LIN {X 0,Y 171.438,Z 260.68,A -85,B 0,C 180,E1 -22896.744,E2 -22896.744} C_VEL
LIN {X 0,Y 171.589,Z 261.495,A -85,B 0,C 180,E1 -22897.442,E2 -22897.442} C_VEL
LIN {X 0,Y 173.16,Z 264.453,A -85,B 0,C 180,E1 -22898.399,E2 -22898.399} C_VEL
LIN {X 0,Y 175.194,Z 266.321,A -85,B 0,C 180,E1 -22899.355,E2 -22899.355} C_VEL
LIN {X 0,Y 177.399,Z 269.743,A -85,B 0,C 180,E1 -22900.432,E2 -22900.432} C_VEL
LIN {X 0,Y 178.724,Z 271.306,A -85,B 0,C 180,E1 -22901.026,E2 -22901.026} C_VEL
LIN {X 0,Y 182.403,Z 276.687,A -85,B 0,C 180,E1 -22902.654,E2 -22902.654} C_VEL
LIN {X 0,Y 187.646,Z 284.442,A -85,B 0,C 180,E1 -22904.791,E2 -22904.791} C_VEL
LIN {X 0,Y 194.854,Z 296.389,A -85,B 0,C 180,E1 -22907.491,E2 -22907.491} C_VEL
LIN {X 0,Y 202.104,Z 310.594,A -85,B 0,C 180,E1 -22910.01,E2 -22910.01} C_VEL
LIN {X 0,Y 211.221,Z 330.235,A -85,B 0,C 180,E1 -22912.895,E2 -22912.895} C_VEL
LIN {X 0,Y 219.903,Z 344.859,A -85,B 0,C 180,E1 -22915.172,E2 -22915.172} C_VEL
LIN {X 0,Y 228.476,Z 356.909,A -85,B 0,C 180,E1 -22917.153,E2 -22917.153} C_VEL
LIN {X 0,Y 236.72,Z 367.005,A -85,B 0,C 180,E1 -22919.009,E2 -22919.009} C_VEL
LIN {X 0,Y 244.162,Z 375.394,A -85,B 0,C 180,E1 -22920.704,E2 -22920.704} C_VEL
LIN {X 0,Y 253.065,Z 384.472,A -85,B 0,C 180,E1 -22922.707,E2 -22922.707} C_VEL
LIN {X 0,Y 263.679,Z 393.909,A -85,B 0,C 180,E1 -22924.986,E2 -22924.986} C_VEL
LIN {X 0,Y 276.755,Z 403.951,A -85,B 0,C 180,E1 -22927.61,E2 -22927.61} C_VEL
LIN {X 0,Y 290.97,Z 414.153,A -85,B 0,C 180,E1 -22930.386,E2 -22930.386} C_VEL
LIN {X 0,Y 299.98,Z 420.738,A -85,B 0,C 180,E1 -22932.268,E2 -22932.268} C_VEL
LIN {X 0,Y 305.133,Z 424.274,A -85,B 0,C 180,E1 -22933.436,E2 -22933.436} C_VEL
LIN {X 0,Y 312.329,Z 429.408,A -85,B 0,C 180,E1 -22935.367,E2 -22935.367} C_VEL
LIN {X 0,Y 318.737,Z 433.404,A -85,B 0,C 180,E1 -22937.262,E2 -22937.262} C_VEL
LIN {X 0,Y 322.774,Z 436.101,A -85,B 0,C 180,E1 -22938.699,E2 -22938.699} C_VEL
LIN {X 0,Y 327.517,Z 439.409,A -85,B 0,C 180,E1 -22940.778,E2 -22940.778} C_VEL
LIN {X 0,Y 331.24,Z 441.589,A -85,B 0,C 180,E1 -22942.686,E2 -22942.686} C_VEL
LIN {X 0,Y 333.408,Z 442.651,A -85,B 0,C 180,E1 -22943.95,E2 -22943.95} C_VEL
LIN {X 0,Y 335.133,Z 443.443,A -85,B 0,C 180,E1 -22945.188,E2 -22945.188} C_VEL
LIN {X 0,Y 336.579,Z 443.963,A -85,B 0,C 180,E1 -22946.409,E2 -22946.409} C_VEL
LIN {X 0,Y 337.607,Z 444.405,A -85,B 0,C 180,E1 -22947.718,E2 -22947.718} C_VEL
LIN {X 0,Y 338.329,Z 444.651,A -85,B 0,C 180,E1 -22950,E2 -22950} C_VEL
LIN {X 0,Y 338.048,Z 444.627,A -85,B 0,C 180,E1 -22951.191,E2 -22951.191} C_VEL
LIN {X 0,Y 337.557,Z 444.334,A -85,B 0,C 180,E1 -22952.386,E2 -22952.386} C_VEL
LIN {X 0,Y 336.548,Z 443.959,A -85,B 0,C 180,E1 -22953.592,E2 -22953.592} C_VEL
LIN {X 0,Y 335.114,Z 443.428,A -85,B 0,C 180,E1 -22954.812,E2 -22954.812} C_VEL
LIN {X 0,Y 332.51,Z 442.258,A -85,B 0,C 180,E1 -22956.593,E2 -22956.593} C_VEL
LIN {X 0,Y 327.517,Z 439.388,A -85,B 0,C 180,E1 -22959.222,E2 -22959.222} C_VEL
LIN {X 0,Y 322.58,Z 435.992,A -85,B 0,C 180,E1 -22961.364,E2 -22961.364} C_VEL
LIN {X 0,Y 318.737,Z 433.444,A -85,B 0,C 180,E1 -22962.738,E2 -22962.738} C_VEL
LIN {X 0,Y 312.33,Z 429.414,A -85,B 0,C 180,E1 -22964.633,E2 -22964.633} C_VEL
LIN {X 0,Y 307.142,Z 425.748,A -85,B 0,C 180,E1 -22966.049,E2 -22966.049} C_VEL
LIN {X 0,Y 301.836,Z 422,A -85,B 0,C 180,E1 -22967.324,E2 -22967.324} C_VEL
LIN {X 0,Y 293.695,Z 416.255,A -85,B 0,C 180,E1 -22969.055,E2 -22969.055} C_VEL
LIN {X 0,Y 282.709,Z 408.344,A -85,B 0,C 180,E1 -22971.217,E2 -22971.217} C_VEL
LIN {X 0,Y 267.705,Z 397.193,A -85,B 0,C 180,E1 -22974.18,E2 -22974.18} C_VEL
LIN {X 0,Y 255.704,Z 386.898,A -85,B 0,C 180,E1 -22976.717,E2 -22976.717} C_VEL
LIN {X 0,Y 247.803,Z 379.333,A -85,B 0,C 180,E1 -22978.456,E2 -22978.456} C_VEL
LIN {X 0,Y 238.025,Z 368.544,A -85,B 0,C 180,E1 -22980.691,E2 -22980.691} C_VEL
LIN {X 0,Y 229.51,Z 358.161,A -85,B 0,C 180,E1 -22982.64,E2 -22982.64} C_VEL
LIN {X 0,Y 221.548,Z 347.302,A -85,B 0,C 180,E1 -22984.436,E2 -22984.436} C_VEL
LIN {X 0,Y 212.624,Z 332.89,A -85,B 0,C 180,E1 -22986.708,E2 -22986.708} C_VEL
LIN {X 0,Y 204.842,Z 316.83,A -85,B 0,C 180,E1 -22989.069,E2 -22989.069} C_VEL
LIN {X 0,Y 200.046,Z 306.438,A -85,B 0,C 180,E1 -22990.683,E2 -22990.683} C_VEL
LIN {X 0,Y 193.65,Z 294.248,A -85,B 0,C 180,E1 -22992.945,E2 -22992.945} C_VEL
LIN {X 0,Y 186.501,Z 282.617,A -85,B 0,C 180,E1 -22995.666,E2 -22995.666} C_VEL
LIN {X 0,Y 180.746,Z 274.26,A -85,B 0,C 180,E1 -22998.065,E2 -22998.065} C_VEL
LIN {X 0,Y 178.122,Z 270.453,A -85,B 0,C 180,E1 -22999.25,E2 -22999.25} C_VEL
LIN {X 0,Y 175.731,Z 267.409,A -85,B 0,C 180,E1 -23000.361,E2 -23000.361} C_VEL
LIN {X 0,Y 174.815,Z 265.84,A -85,B 0,C 180,E1 -23000.828,E2 -23000.828} C_VEL
LIN {X 0,Y 172.55,Z 263.632,A -85,B 0,C 180,E1 -23001.914,E2 -23001.914} C_VEL
LIN {X 0,Y 171.504,Z 261.178,A -85,B 0,C 180,E1 -23002.721,E2 -23002.721} C_VEL
LIN {X 0,Y 171.432,Z 260.639,A -85,B 0,C 180,E1 -23003.529,E2 -23003.529} C_VEL
LIN {X 0,Y 171.454,Z 260.623,A -85,B 0,C 180,E1 -23009.406,E2 -23009.406} C_VEL
LIN {X 0,Y 171.456,Z 260.598,A -85,B 0,C 180,E1 -23014.393,E2 -23014.393} C_VEL
LIN {X 0,Y 171.576,Z 260.565,A -85,B 0,C 180,E1 -23020.873,E2 -23020.873} C_VEL
LIN {X 0,Y 171.591,Z 260.61,A -85,B 0,C 180,E1 -23025.775,E2 -23025.775} C_VEL
LIN {X 0,Y 171.85,Z 260.526,A -85,B 0,C 180,E1 -23030.586,E2 -23030.586} C_VEL
LIN {X 0,Y 171.819,Z 260.581,A -85,B 0,C 180,E1 -23035.309,E2 -23035.309} C_VEL
LIN {X 0,Y 172.331,Z 260.463,A -85,B 0,C 180,E1 -23040.001,E2 -23040.001} C_VEL
LIN {X 0,Y 171.81,Z 260.584,A -85,B 0,C 180,E1 -23044.694,E2 -23044.694} C_VEL
LIN {X 0,Y 171.844,Z 260.524,A -85,B 0,C 180,E1 -23049.417,E2 -23049.417} C_VEL
LIN {X 0,Y 171.569,Z 260.611,A -85,B 0,C 180,E1 -23054.229,E2 -23054.229} C_VEL
LIN {X 0,Y 171.543,Z 260.569,A -85,B 0,C 180,E1 -23059.56,E2 -23059.56} C_VEL
LIN {X 0,Y 171.463,Z 260.59,A -85,B 0,C 180,E1 -23065.612,E2 -23065.612} C_VEL
LIN {X 0,Y 171.458,Z 260.628,A -85,B 0,C 180,E1 -23070.596,E2 -23070.596} C_VEL
LIN {X 0,Y 171.405,Z 260.744,A -85,B 0,C 180,E1 -23076.39,E2 -23076.39} C_VEL
LIN {X 0,Y 171.537,Z 261.477,A -85,B 0,C 180,E1 -23076.997,E2 -23076.997} C_VEL
LIN {X 0,Y 173.009,Z 264.327,A -85,B 0,C 180,E1 -23077.946,E2 -23077.946} C_VEL
LIN {X 0,Y 175.541,Z 267.445,A -85,B 0,C 180,E1 -23079.183,E2 -23079.183} C_VEL
LIN {X 0,Y 178.493,Z 271.992,A -85,B 0,C 180,E1 -23080.599,E2 -23080.599} C_VEL
LIN {X 0,Y 182.943,Z 279.543,A -85,B 0,C 180,E1 -23082.618,E2 -23082.618} C_VEL
LIN {X 0,Y 189.539,Z 291.631,A -85,B 0,C 180,E1 -23085.361,E2 -23085.361} C_VEL
LIN {X 0,Y 194.252,Z 301.668,A -85,B 0,C 180,E1 -23087.205,E2 -23087.205} C_VEL
LIN {X 0,Y 199.621,Z 314.742,A -85,B 0,C 180,E1 -23089.216,E2 -23089.216} C_VEL
LIN {X 0,Y 201.158,Z 324.413,A -85,B 0,C 180,E1 -23090.032,E2 -23090.032} C_VEL
LIN {X 0,Y 201.394,Z 328.625,A -85,B 0,C 180,E1 -23090.279,E2 -23090.279} C_VEL
LIN {X 0,Y 199.139,Z 368.462,A -85,B 0,C 180,E1 -23091.638,E2 -23091.638} C_VEL
LIN {X 0,Y 197.78,Z 380.363,A -85,B 0,C 180,E1 -23092.301,E2 -23092.301} C_VEL
LIN {X 0,Y 195.345,Z 393.909,A -85,B 0,C 180,E1 -23093.425,E2 -23093.425} C_VEL
LIN {X 0,Y 192.883,Z 404.427,A -85,B 0,C 180,E1 -23094.66,E2 -23094.66} C_VEL
LIN {X 0,Y 190.357,Z 413.699,A -85,B 0,C 180,E1 -23096.054,E2 -23096.054} C_VEL
LIN {X 0,Y 187.599,Z 422.641,A -85,B 0,C 180,E1 -23097.734,E2 -23097.734} C_VEL
LIN {X 0,Y 184.625,Z 431.165,A -85,B 0,C 180,E1 -23099.71,E2 -23099.71} C_VEL
LIN {X 0,Y 181.879,Z 438.38,A -85,B 0,C 180,E1 -23101.748,E2 -23101.748} C_VEL
LIN {X 0,Y 179.461,Z 444.58,A -85,B 0,C 180,E1 -23103.86,E2 -23103.86} C_VEL
LIN {X 0,Y 176.889,Z 451.12,A -85,B 0,C 180,E1 -23106.59,E2 -23106.59} C_VEL
LIN {X 0,Y 174.917,Z 455.619,A -85,B 0,C 180,E1 -23108.801,E2 -23108.801} C_VEL
LIN {X 0,Y 172.575,Z 461.112,A -85,B 0,C 180,E1 -23112.216,E2 -23112.216} C_VEL
LIN {X 0,Y 170.821,Z 465.44,A -85,B 0,C 180,E1 -23115.709,E2 -23115.709} C_VEL
LIN {X 0,Y 170.017,Z 467.812,A -85,B 0,C 180,E1 -23118.072,E2 -23118.072} C_VEL
LIN {X 0,Y 169.418,Z 469.615,A -85,B 0,C 180,E1 -23120.449,E2 -23120.449} C_VEL
LIN {X 0,Y 168.933,Z 472.074,A -85,B 0,C 180,E1 -23125.227,E2 -23125.227} C_VEL
LIN {X 0,Y 168.87,Z 472.72,A -85,B 0,C 180,E1 -23128.402,E2 -23128.402} C_VEL
LIN {X 0,Y 168.968,Z 472.826,A -85,B 0,C 180,E1 -23130,E2 -23130} C_VEL
LIN {X 0,Y 168.853,Z 472.607,A -85,B 0,C 180,E1 -23132.627,E2 -23132.627} C_VEL
LIN {X 0,Y 168.863,Z 472.072,A -85,B 0,C 180,E1 -23134.775,E2 -23134.775} C_VEL
LIN {X 0,Y 169.207,Z 470.166,A -85,B 0,C 180,E1 -23138.609,E2 -23138.609} C_VEL
LIN {X 0,Y 168.941,Z 468.894,A -85,B 0,C 180,E1 -23140.562,E2 -23140.562} C_VEL
LIN {X 0,Y 167.041,Z 466.261,A -85,B 0,C 180,E1 -23143.759,E2 -23143.759} C_VEL
LIN {X 0,Y 165.575,Z 462.945,A -85,B 0,C 180,E1 -23146.944,E2 -23146.944} C_VEL
LIN {X 0,Y 165.989,Z 460.535,A -85,B 0,C 180,E1 -23148.811,E2 -23148.811} C_VEL
LIN {X 0,Y 168.79,Z 454.39,A -85,B 0,C 180,E1 -23152.653,E2 -23152.653} C_VEL
LIN {X 0,Y 171.612,Z 447.998,A -85,B 0,C 180,E1 -23155.712,E2 -23155.712} C_VEL
LIN {X 0,Y 174.325,Z 441.439,A -85,B 0,C 180,E1 -23158.275,E2 -23158.275} C_VEL
LIN {X 0,Y 177.779,Z 432.89,A -85,B 0,C 180,E1 -23160.925,E2 -23160.925} C_VEL
LIN {X 0,Y 180.808,Z 424.715,A -85,B 0,C 180,E1 -23162.968,E2 -23162.968} C_VEL
LIN {X 0,Y 183.683,Z 416.208,A -85,B 0,C 180,E1 -23164.69,E2 -23164.69} C_VEL
LIN {X 0,Y 186.22,Z 407.495,A -85,B 0,C 180,E1 -23166.135,E2 -23166.135} C_VEL
LIN {X 0,Y 188.779,Z 397.743,A -85,B 0,C 180,E1 -23167.394,E2 -23167.394} C_VEL
LIN {X 0,Y 190.909,Z 387.666,A -85,B 0,C 180,E1 -23168.405,E2 -23168.405} C_VEL
LIN {X 0,Y 192.614,Z 377.207,A -85,B 0,C 180,E1 -23169.182,E2 -23169.182} C_VEL
LIN {X 0,Y 193.75,Z 367.131,A -85,B 0,C 180,E1 -23169.702,E2 -23169.702} C_VEL
LIN {X 0,Y 195.936,Z 327.052,A -85,B 0,C 180,E1 -23171.126,E2 -23171.126} C_VEL
LIN {X 0,Y 194.539,Z 317.878,A -85,B 0,C 180,E1 -23171.927,E2 -23171.927} C_VEL
LIN {X 0,Y 189.037,Z 304.24,A -85,B 0,C 180,E1 -23174.133,E2 -23174.133} C_VEL
LIN {X 0,Y 184.476,Z 294.52,A -85,B 0,C 180,E1 -23176.044,E2 -23176.044} C_VEL
LIN {X 0,Y 177.798,Z 282.073,A -85,B 0,C 180,E1 -23179.051,E2 -23179.051} C_VEL
LIN {X 0,Y 173.97,Z 275.954,A -85,B 0,C 180,E1 -23180.905,E2 -23180.905} C_VEL
LIN {X 0,Y 171.06,Z 271.361,A -85,B 0,C 180,E1 -23182.419,E2 -23182.419} C_VEL
LIN {X 0,Y 168.608,Z 267.983,A -85,B 0,C 180,E1 -23183.744,E2 -23183.744} C_VEL
LIN {X 0,Y 167.771,Z 266.738,A -85,B 0,C 180,E1 -23184.222,E2 -23184.222} C_VEL
LIN {X 0,Y 165.529,Z 264.614,A -85,B 0,C 180,E1 -23185.464,E2 -23185.464} C_VEL
LIN {X 0,Y 164.434,Z 262.097,A -85,B 0,C 180,E1 -23186.419,E2 -23186.419} C_VEL
LIN {X 0,Y 164.371,Z 261.527,A -85,B 0,C 180,E1 -23187.272,E2 -23187.272} C_VEL
LIN {X 0,Y 164.341,Z 261.476,A -85,B 0,C 180,E1 -23191.937,E2 -23191.937} C_VEL
LIN {X 0,Y 164.412,Z 261.47,A -85,B 0,C 180,E1 -23194.692,E2 -23194.692} C_VEL
LIN {X 0,Y 164.486,Z 261.449,A -85,B 0,C 180,E1 -23200.05,E2 -23200.05} C_VEL
LIN {X 0,Y 164.499,Z 261.486,A -85,B 0,C 180,E1 -23205.146,E2 -23205.146} C_VEL
LIN {X 0,Y 164.765,Z 261.405,A -85,B 0,C 180,E1 -23210.175,E2 -23210.175} C_VEL
LIN {X 0,Y 164.825,Z 261.412,A -85,B 0,C 180,E1 -23212.649,E2 -23212.649} C_VEL
LIN {X 0,Y 165.045,Z 261.392,A -85,B 0,C 180,E1 -23217.558,E2 -23217.558} C_VEL
LIN {X 0,Y 165.293,Z 261.339,A -85,B 0,C 180,E1 -23219.999,E2 -23219.999} C_VEL
LIN {X 0,Y 164.768,Z 261.461,A -85,B 0,C 180,E1 -23224.892,E2 -23224.892} C_VEL
LIN {X 0,Y 164.834,Z 261.419,A -85,B 0,C 180,E1 -23227.347,E2 -23227.347} C_VEL
LIN {X 0,Y 164.703,Z 261.418,A -85,B 0,C 180,E1 -23231.061,E2 -23231.061} C_VEL
LIN {X 0,Y 164.54,Z 261.49,A -85,B 0,C 180,E1 -23234.848,E2 -23234.848} C_VEL
LIN {X 0,Y 164.471,Z 261.452,A -85,B 0,C 180,E1 -23239.988,E2 -23239.988} C_VEL
LIN {X 0,Y 164.383,Z 261.473,A -85,B 0,C 180,E1 -23246.127,E2 -23246.127} C_VEL
LIN {X 0,Y 164.385,Z 261.491,A -85,B 0,C 180,E1 -23252.376,E2 -23252.376} C_VEL
LIN {X 0,Y 164.377,Z 261.818,A -85,B 0,C 180,E1 -23253.765,E2 -23253.765} C_VEL
LIN {X 0,Y 164.717,Z 263.033,A -85,B 0,C 180,E1 -23254.365,E2 -23254.365} C_VEL
LIN {X 0,Y 166.416,Z 265.672,A -85,B 0,C 180,E1 -23255.434,E2 -23255.434} C_VEL
LIN {X 0,Y 168.281,Z 267.143,A -85,B 0,C 180,E1 -23256.427,E2 -23256.427} C_VEL
LIN {X 0,Y 170.322,Z 270.482,A -85,B 0,C 180,E1 -23257.582,E2 -23257.582} C_VEL
LIN {X 0,Y 172.089,Z 272.336,A -85,B 0,C 180,E1 -23258.467,E2 -23258.467} C_VEL
LIN {X 0,Y 174.73,Z 276.02,A -85,B 0,C 180,E1 -23259.785,E2 -23259.785} C_VEL
LIN {X 0,Y 181.065,Z 285.342,A -85,B 0,C 180,E1 -23262.689,E2 -23262.689} C_VEL
LIN {X 0,Y 187.19,Z 295.122,A -85,B 0,C 180,E1 -23265.219,E2 -23265.219} C_VEL
LIN {X 0,Y 192.958,Z 305.583,A -85,B 0,C 180,E1 -23267.427,E2 -23267.427} C_VEL
LIN {X 0,Y 199.509,Z 319.465,A -85,B 0,C 180,E1 -23269.79,E2 -23269.79} C_VEL
LIN {X 0,Y 206.442,Z 334.522,A -85,B 0,C 180,E1 -23272.063,E2 -23272.063} C_VEL
LIN {X 0,Y 215.092,Z 349.3,A -85,B 0,C 180,E1 -23274.448,E2 -23274.448} C_VEL
LIN {X 0,Y 223.821,Z 361.843,A -85,B 0,C 180,E1 -23276.619,E2 -23276.619} C_VEL
LIN {X 0,Y 233.68,Z 374.129,A -85,B 0,C 180,E1 -23279.106,E2 -23279.106} C_VEL
LIN {X 0,Y 244.415,Z 385.978,A -85,B 0,C 180,E1 -23281.798,E2 -23281.798} C_VEL
LIN {X 0,Y 255.3,Z 396.076,A -85,B 0,C 180,E1 -23284.361,E2 -23284.361} C_VEL
LIN {X 0,Y 267.258,Z 405.597,A -85,B 0,C 180,E1 -23286.98,E2 -23286.98} C_VEL
LIN {X 0,Y 280.847,Z 415.193,A -85,B 0,C 180,E1 -23289.782,E2 -23289.782} C_VEL
LIN {X 0,Y 289.662,Z 421.381,A -85,B 0,C 180,E1 -23291.614,E2 -23291.614} C_VEL
LIN {X 0,Y 298.799,Z 427.73,A -85,B 0,C 180,E1 -23293.606,E2 -23293.606} C_VEL
LIN {X 0,Y 305.423,Z 432.473,A -85,B 0,C 180,E1 -23295.338,E2 -23295.338} C_VEL
LIN {X 0,Y 311.032,Z 436.104,A -85,B 0,C 180,E1 -23296.941,E2 -23296.941} C_VEL
LIN {X 0,Y 315.717,Z 438.976,A -85,B 0,C 180,E1 -23298.443,E2 -23298.443} C_VEL
LIN {X 0,Y 320.624,Z 442.508,A -85,B 0,C 180,E1 -23300.531,E2 -23300.531} C_VEL
LIN {X 0,Y 324.682,Z 444.989,A -85,B 0,C 180,E1 -23302.538,E2 -23302.538} C_VEL
LIN {X 0,Y 326.954,Z 446.165,A -85,B 0,C 180,E1 -23303.83,E2 -23303.83} C_VEL
LIN {X 0,Y 328.836,Z 447.066,A -85,B 0,C 180,E1 -23305.096,E2 -23305.096} C_VEL
LIN {X 0,Y 330.825,Z 447.822,A -85,B 0,C 180,E1 -23306.805,E2 -23306.805} C_VEL
LIN {X 0,Y 331.953,Z 448.338,A -85,B 0,C 180,E1 -23308.787,E2 -23308.787} C_VEL
LIN {X 0,Y 332.279,Z 448.347,A -85,B 0,C 180,E1 -23310,E2 -23310} C_VEL
LIN {X 0,Y 331.971,Z 448.319,A -85,B 0,C 180,E1 -23311.213,E2 -23311.213} C_VEL
LIN {X 0,Y 331.432,Z 448.026,A -85,B 0,C 180,E1 -23312.431,E2 -23312.431} C_VEL
LIN {X 0,Y 330.339,Z 447.637,A -85,B 0,C 180,E1 -23313.659,E2 -23313.659} C_VEL
LIN {X 0,Y 328.819,Z 447.054,A -85,B 0,C 180,E1 -23314.904,E2 -23314.904} C_VEL
LIN {X 0,Y 325.667,Z 445.509,A -85,B 0,C 180,E1 -23316.937,E2 -23316.937} C_VEL
LIN {X 0,Y 322.096,Z 443.445,A -85,B 0,C 180,E1 -23318.786,E2 -23318.786} C_VEL
LIN {X 0,Y 319.098,Z 441.471,A -85,B 0,C 180,E1 -23320.148,E2 -23320.148} C_VEL
LIN {X 0,Y 315.637,Z 438.998,A -85,B 0,C 180,E1 -23321.566,E2 -23321.566} C_VEL
LIN {X 0,Y 310.43,Z 435.777,A -85,B 0,C 180,E1 -23323.224,E2 -23323.224} C_VEL
LIN {X 0,Y 305.196,Z 432.342,A -85,B 0,C 180,E1 -23324.726,E2 -23324.726} C_VEL
LIN {X 0,Y 298.774,Z 427.714,A -85,B 0,C 180,E1 -23326.396,E2 -23326.396} C_VEL
LIN {X 0,Y 289.619,Z 421.383,A -85,B 0,C 180,E1 -23328.389,E2 -23328.389} C_VEL
LIN {X 0,Y 278.513,Z 413.636,A -85,B 0,C 180,E1 -23330.688,E2 -23330.688} C_VEL
LIN {X 0,Y 265.442,Z 404.273,A -85,B 0,C 180,E1 -23333.4,E2 -23333.4} C_VEL
LIN {X 0,Y 252.686,Z 393.803,A -85,B 0,C 180,E1 -23336.239,E2 -23336.239} C_VEL
LIN {X 0,Y 242.681,Z 384.19,A -85,B 0,C 180,E1 -23338.632,E2 -23338.632} C_VEL
LIN {X 0,Y 231.94,Z 372.072,A -85,B 0,C 180,E1 -23341.336,E2 -23341.336} C_VEL
LIN {X 0,Y 222.059,Z 359.477,A -85,B 0,C 180,E1 -23343.822,E2 -23343.822} C_VEL
LIN {X 0,Y 212.255,Z 344.794,A -85,B 0,C 180,E1 -23346.29,E2 -23346.29} C_VEL
LIN {X 0,Y 204.9,Z 331.451,A -85,B 0,C 180,E1 -23348.411,E2 -23348.411} C_VEL
LIN {X 0,Y 195.717,Z 311.251,A -85,B 0,C 180,E1 -23351.556,E2 -23351.556} C_VEL
LIN {X 0,Y 189.608,Z 299.314,A -85,B 0,C 180,E1 -23353.839,E2 -23353.839} C_VEL
LIN {X 0,Y 182.777,Z 287.906,A -85,B 0,C 180,E1 -23356.584,E2 -23356.584} C_VEL
LIN {X 0,Y 176.826,Z 279.161,A -85,B 0,C 180,E1 -23359.209,E2 -23359.209} C_VEL
LIN {X 0,Y 174.486,Z 275.766,A -85,B 0,C 180,E1 -23360.328,E2 -23360.328} C_VEL
LIN {X 0,Y 171.432,Z 271.566,A -85,B 0,C 180,E1 -23361.863,E2 -23361.863} C_VEL
LIN {X 0,Y 169.042,Z 268.695,A -85,B 0,C 180,E1 -23363.114,E2 -23363.114} C_VEL
LIN {X 0,Y 167.925,Z 266.813,A -85,B 0,C 180,E1 -23363.762,E2 -23363.762} C_VEL
LIN {X 0,Y 165.577,Z 264.662,A -85,B 0,C 180,E1 -23365.054,E2 -23365.054} C_VEL
LIN {X 0,Y 164.44,Z 262.027,A -85,B 0,C 180,E1 -23366.04,E2 -23366.04} C_VEL
LIN {X 0,Y 164.345,Z 261.512,A -85,B 0,C 180,E1 -23366.924,E2 -23366.924} C_VEL
LIN {X 0,Y 164.401,Z 261.505,A -85,B 0,C 180,E1 -23369.139,E2 -23369.139} C_VEL
LIN {X 0,Y 164.404,Z 261.479,A -85,B 0,C 180,E1 -23374.694,E2 -23374.694} C_VEL
LIN {X 0,Y 164.483,Z 261.45,A -85,B 0,C 180,E1 -23380.053,E2 -23380.053} C_VEL
LIN {X 0,Y 164.54,Z 261.49,A -85,B 0,C 180,E1 -23385.152,E2 -23385.152} C_VEL
LIN {X 0,Y 164.769,Z 261.406,A -85,B 0,C 180,E1 -23390.178,E2 -23390.178} C_VEL
LIN {X 0,Y 164.834,Z 261.419,A -85,B 0,C 180,E1 -23392.653,E2 -23392.653} C_VEL
LIN {X 0,Y 165.049,Z 261.384,A -85,B 0,C 180,E1 -23397.561,E2 -23397.561} C_VEL
LIN {X 0,Y 165.293,Z 261.339,A -85,B 0,C 180,E1 -23400.001,E2 -23400.001} C_VEL
LIN {X 0,Y 164.759,Z 261.462,A -85,B 0,C 180,E1 -23404.895,E2 -23404.895} C_VEL
LIN {X 0,Y 164.825,Z 261.412,A -85,B 0,C 180,E1 -23407.351,E2 -23407.351} C_VEL
LIN {X 0,Y 164.702,Z 261.419,A -85,B 0,C 180,E1 -23411.06,E2 -23411.06} C_VEL
LIN {X 0,Y 164.477,Z 261.45,A -85,B 0,C 180,E1 -23417.405,E2 -23417.405} C_VEL
LIN {X 0,Y 164.475,Z 261.451,A -85,B 0,C 180,E1 -23419.99,E2 -23419.99} C_VEL
LIN {X 0,Y 164.39,Z 261.467,A -85,B 0,C 180,E1 -23426.131,E2 -23426.131} C_VEL
LIN {X 0,Y 164.387,Z 261.5,A -85,B 0,C 180,E1 -23432.379,E2 -23432.379} C_VEL
LIN {X 0,Y 164.408,Z 261.87,A -85,B 0,C 180,E1 -23433.413,E2 -23433.413} C_VEL
LIN {X 0,Y 164.782,Z 263.221,A -85,B 0,C 180,E1 -23434.037,E2 -23434.037} C_VEL
LIN {X 0,Y 166.488,Z 265.738,A -85,B 0,C 180,E1 -23435.092,E2 -23435.092} C_VEL
LIN {X 0,Y 168.285,Z 267.309,A -85,B 0,C 180,E1 -23436.059,E2 -23436.059} C_VEL
LIN {X 0,Y 170.455,Z 270.69,A -85,B 0,C 180,E1 -23437.272,E2 -23437.272} C_VEL
LIN {X 0,Y 172.379,Z 273.331,A -85,B 0,C 180,E1 -23438.273,E2 -23438.273} C_VEL
LIN {X 0,Y 176.106,Z 279.391,A -85,B 0,C 180,E1 -23440.15,E2 -23440.15} C_VEL
LIN {X 0,Y 180.45,Z 286.862,A -85,B 0,C 180,E1 -23442.182,E2 -23442.182} C_VEL
LIN {X 0,Y 187.19,Z 300.02,A -85,B 0,C 180,E1 -23445.097,E2 -23445.097} C_VEL
LIN {X 0,Y 193.374,Z 314.666,A -85,B 0,C 180,E1 -23447.607,E2 -23447.607} C_VEL
LIN {X 0,Y 194.788,Z 318.831,A -85,B 0,C 180,E1 -23448.185,E2 -23448.185} C_VEL
LIN {X 0,Y 195.976,Z 327.581,A -85,B 0,C 180,E1 -23448.909,E2 -23448.909} C_VEL
LIN {X 0,Y 193.642,Z 368.059,A -85,B 0,C 180,E1 -23450.324,E2 -23450.324} C_VEL
LIN {X 0,Y 192.322,Z 379.414,A -85,B 0,C 180,E1 -23450.96,E2 -23450.96} C_VEL
LIN {X 0,Y 190.199,Z 391.526,A -85,B 0,C 180,E1 -23451.931,E2 -23451.931} C_VEL
LIN {X 0,Y 187.141,Z 404.234,A -85,B 0,C 180,E1 -23453.403,E2 -23453.403} C_VEL
LIN {X 0,Y 184.509,Z 413.506,A -85,B 0,C 180,E1 -23454.822,E2 -23454.822} C_VEL
LIN {X 0,Y 181.606,Z 422.447,A -85,B 0,C 180,E1 -23456.533,E2 -23456.533} C_VEL
LIN {X 0,Y 178.5,Z 430.971,A -85,B 0,C 180,E1 -23458.555,E2 -23458.555} C_VEL
LIN {X 0,Y 175.634,Z 438.186,A -85,B 0,C 180,E1 -23460.648,E2 -23460.648} C_VEL
LIN {X 0,Y 173.083,Z 444.387,A -85,B 0,C 180,E1 -23462.819,E2 -23462.819} C_VEL
LIN {X 0,Y 170.371,Z 450.927,A -85,B 0,C 180,E1 -23465.637,E2 -23465.637} C_VEL
LIN {X 0,Y 168.291,Z 455.426,A -85,B 0,C 180,E1 -23467.923,E2 -23467.923} C_VEL
LIN {X 0,Y 165.816,Z 460.919,A -85,B 0,C 180,E1 -23471.465,E2 -23471.465} C_VEL
LIN {X 0,Y 163.898,Z 465.246,A -85,B 0,C 180,E1 -23475.091,E2 -23475.091} C_VEL
LIN {X 0,Y 163.049,Z 467.618,A -85,B 0,C 180,E1 -23477.554,E2 -23477.554} C_VEL
LIN {X 0,Y 162.399,Z 469.422,A -85,B 0,C 180,E1 -23480.032,E2 -23480.032} C_VEL
LIN {X 0,Y 161.851,Z 471.881,A -85,B 0,C 180,E1 -23485.018,E2 -23485.018} C_VEL
LIN {X 0,Y 161.8,Z 472.475,A -85,B 0,C 180,E1 -23487.511,E2 -23487.511} C_VEL
LIN {X 0,Y 161.884,Z 472.634,A -85,B 0,C 180,E1 -23490,E2 -23490} C_VEL
LIN {X 0,Y 161.763,Z 472.474,A -85,B 0,C 180,E1 -23492.49,E2 -23492.49} C_VEL
LIN {X 0,Y 161.767,Z 471.879,A -85,B 0,C 180,E1 -23494.985,E2 -23494.985} C_VEL
LIN {X 0,Y 162.377,Z 469.421,A -85,B 0,C 180,E1 -23499.97,E2 -23499.97} C_VEL
LIN {X 0,Y 163.451,Z 466.465,A -85,B 0,C 180,E1 -23503.679,E2 -23503.679} C_VEL
LIN {X 0,Y 165.062,Z 462.472,A -85,B 0,C 180,E1 -23507.34,E2 -23507.34} C_VEL
LIN {X 0,Y 165.989,Z 460.535,A -85,B 0,C 180,E1 -23508.811,E2 -23508.811} C_VEL
LIN {X 0,Y 166.546,Z 457.94,A -85,B 0,C 180,E1 -23510.63,E2 -23510.63} C_VEL
LIN {X 0,Y 165.954,Z 453.279,A -85,B 0,C 180,E1 -23513.643,E2 -23513.643} C_VEL
LIN {X 0,Y 165.647,Z 448.122,A -85,B 0,C 180,E1 -23516.562,E2 -23516.562} C_VEL
LIN {X 0,Y 166.624,Z 444.506,A -85,B 0,C 180,E1 -23518.171,E2 -23518.171} C_VEL
LIN {X 0,Y 170.2,Z 436.367,A -85,B 0,C 180,E1 -23521.075,E2 -23521.075} C_VEL
LIN {X 0,Y 174.476,Z 425.656,A -85,B 0,C 180,E1 -23523.979,E2 -23523.979} C_VEL
LIN {X 0,Y 177.469,Z 417.367,A -85,B 0,C 180,E1 -23525.741,E2 -23525.741} C_VEL
LIN {X 0,Y 180.541,Z 407.303,A -85,B 0,C 180,E1 -23527.462,E2 -23527.462} C_VEL
LIN {X 0,Y 183.202,Z 397.551,A -85,B 0,C 180,E1 -23528.739,E2 -23528.739} C_VEL
LIN {X 0,Y 185.139,Z 388.76,A -85,B 0,C 180,E1 -23529.659,E2 -23529.659} C_VEL
LIN {X 0,Y 187.025,Z 378.084,A -85,B 0,C 180,E1 -23530.483,E2 -23530.483} C_VEL
LIN {X 0,Y 188.275,Z 367.782,A -85,B 0,C 180,E1 -23531.043,E2 -23531.043} C_VEL
LIN {X 0,Y 190.572,Z 328.375,A -85,B 0,C 180,E1 -23532.474,E2 -23532.474} C_VEL
LIN {X 0,Y 189.458,Z 320.684,A -85,B 0,C 180,E1 -23533.17,E2 -23533.17} C_VEL
LIN {X 0,Y 183.649,Z 306.172,A -85,B 0,C 180,E1 -23535.67,E2 -23535.67} C_VEL
LIN {X 0,Y 178.643,Z 295.698,A -85,B 0,C 180,E1 -23537.937,E2 -23537.937} C_VEL
LIN {X 0,Y 173.44,Z 286.121,A -85,B 0,C 180,E1 -23540.469,E2 -23540.469} C_VEL
LIN {X 0,Y 170.39,Z 281.039,A -85,B 0,C 180,E1 -23542.059,E2 -23542.059} C_VEL
LIN {X 0,Y 167.856,Z 276.923,A -85,B 0,C 180,E1 -23543.462,E2 -23543.462} C_VEL
LIN {X 0,Y 165.358,Z 273.352,A -85,B 0,C 180,E1 -23544.901,E2 -23544.901} C_VEL
LIN {X 0,Y 162.366,Z 269.939,A -85,B 0,C 180,E1 -23546.688,E2 -23546.688} C_VEL
LIN {X 0,Y 161.145,Z 267.827,A -85,B 0,C 180,E1 -23547.52,E2 -23547.52} C_VEL
LIN {X 0,Y 158.817,Z 265.891,A -85,B 0,C 180,E1 -23549.019,E2 -23549.019} C_VEL
LIN {X 0,Y 157.382,Z 262.956,A -85,B 0,C 180,E1 -23550.394,E2 -23550.394} C_VEL
LIN {X 0,Y 157.296,Z 262.41,A -85,B 0,C 180,E1 -23551.294,E2 -23551.294} C_VEL
LIN {X 0,Y 157.31,Z 262.376,A -85,B 0,C 180,E1 -23556.29,E2 -23556.29} C_VEL
LIN {X 0,Y 157.406,Z 262.326,A -85,B 0,C 180,E1 -23561.786,E2 -23561.786} C_VEL
LIN {X 0,Y 157.513,Z 262.34,A -85,B 0,C 180,E1 -23567.108,E2 -23567.108} C_VEL
LIN {X 0,Y 157.687,Z 262.287,A -85,B 0,C 180,E1 -23569.729,E2 -23569.729} C_VEL
LIN {X 0,Y 157.762,Z 262.286,A -85,B 0,C 180,E1 -23572.318,E2 -23572.318} C_VEL
LIN {X 0,Y 158.256,Z 262.214,A -85,B 0,C 180,E1 -23579.999,E2 -23579.999} C_VEL
LIN {X 0,Y 157.77,Z 262.292,A -85,B 0,C 180,E1 -23587.678,E2 -23587.678} C_VEL
LIN {X 0,Y 157.637,Z 262.298,A -85,B 0,C 180,E1 -23591.237,E2 -23591.237} C_VEL
LIN {X 0,Y 157.469,Z 262.359,A -85,B 0,C 180,E1 -23595.531,E2 -23595.531} C_VEL
LIN {X 0,Y 157.366,Z 262.343,A -85,B 0,C 180,E1 -23600.932,E2 -23600.932} C_VEL
LIN {X 0,Y 157.308,Z 262.351,A -85,B 0,C 180,E1 -23606.68,E2 -23606.68} C_VEL
LIN {X 0,Y 157.331,Z 262.676,A -85,B 0,C 180,E1 -23609.705,E2 -23609.705} C_VEL
LIN {X 0,Y 157.682,Z 263.84,A -85,B 0,C 180,E1 -23610.462,E2 -23610.462} C_VEL
LIN {X 0,Y 159.304,Z 266.469,A -85,B 0,C 180,E1 -23611.7,E2 -23611.7} C_VEL
LIN {X 0,Y 161.55,Z 268.344,A -85,B 0,C 180,E1 -23613.126,E2 -23613.126} C_VEL
LIN {X 0,Y 163.611,Z 271.568,A -85,B 0,C 180,E1 -23614.472,E2 -23614.472} C_VEL
LIN {X 0,Y 165.519,Z 273.546,A -85,B 0,C 180,E1 -23615.574,E2 -23615.574} C_VEL
LIN {X 0,Y 168.084,Z 277.121,A -85,B 0,C 180,E1 -23617.037,E2 -23617.037} C_VEL
LIN {X 0,Y 169.495,Z 279.002,A -85,B 0,C 180,E1 -23617.797,E2 -23617.797} C_VEL
LIN {X 0,Y 172.426,Z 283.14,A -85,B 0,C 180,E1 -23619.313,E2 -23619.313} C_VEL
LIN {X 0,Y 177.321,Z 290.463,A -85,B 0,C 180,E1 -23621.66,E2 -23621.66} C_VEL
LIN {X 0,Y 183.081,Z 299.863,A -85,B 0,C 180,E1 -23624.183,E2 -23624.183} C_VEL
LIN {X 0,Y 188.608,Z 310.114,A -85,B 0,C 180,E1 -23626.427,E2 -23626.427} C_VEL
LIN {X 0,Y 194.311,Z 322.366,A -85,B 0,C 180,E1 -23628.613,E2 -23628.613} C_VEL
LIN {X 0,Y 201.691,Z 338.776,A -85,B 0,C 180,E1 -23631.187,E2 -23631.187} C_VEL
LIN {X 0,Y 210.204,Z 353.586,A -85,B 0,C 180,E1 -23633.662,E2 -23633.662} C_VEL
LIN {X 0,Y 218.124,Z 365.416,A -85,B 0,C 180,E1 -23635.857,E2 -23635.857} C_VEL
LIN {X 0,Y 226.087,Z 375.932,A -85,B 0,C 180,E1 -23638.099,E2 -23638.099} C_VEL
LIN {X 0,Y 234.414,Z 385.578,A -85,B 0,C 180,E1 -23640.393,E2 -23640.393} C_VEL
LIN {X 0,Y 242.797,Z 394.301,A -85,B 0,C 180,E1 -23642.631,E2 -23642.631} C_VEL
LIN {X 0,Y 253.56,Z 403.723,A -85,B 0,C 180,E1 -23645.288,E2 -23645.288} C_VEL
LIN {X 0,Y 265.351,Z 412.559,A -85,B 0,C 180,E1 -23647.969,E2 -23647.969} C_VEL
LIN {X 0,Y 278.845,Z 421.692,A -85,B 0,C 180,E1 -23650.874,E2 -23650.874} C_VEL
LIN {X 0,Y 289.824,Z 429.138,A -85,B 0,C 180,E1 -23653.299,E2 -23653.299} C_VEL
LIN {X 0,Y 296.497,Z 433.769,A -85,B 0,C 180,E1 -23654.886,E2 -23654.886} C_VEL
LIN {X 0,Y 303.254,Z 438.417,A -85,B 0,C 180,E1 -23656.742,E2 -23656.742} C_VEL
LIN {X 0,Y 309.806,Z 442.445,A -85,B 0,C 180,E1 -23658.772,E2 -23658.772} C_VEL
LIN {X 0,Y 315.026,Z 446.149,A -85,B 0,C 180,E1 -23661.016,E2 -23661.016} C_VEL
LIN {X 0,Y 318.729,Z 448.42,A -85,B 0,C 180,E1 -23662.857,E2 -23662.857} C_VEL
LIN {X 0,Y 322.204,Z 450.145,A -85,B 0,C 180,E1 -23664.995,E2 -23664.995} C_VEL
LIN {X 0,Y 323.942,Z 450.874,A -85,B 0,C 180,E1 -23666.345,E2 -23666.345} C_VEL
LIN {X 0,Y 325.024,Z 451.295,A -85,B 0,C 180,E1 -23667.521,E2 -23667.521} C_VEL
LIN {X 0,Y 325.635,Z 451.587,A -85,B 0,C 180,E1 -23668.763,E2 -23668.763} C_VEL
LIN {X 0,Y 325.967,Z 451.615,A -85,B 0,C 180,E1 -23670,E2 -23670} C_VEL
LIN {X 0,Y 325.651,Z 451.573,A -85,B 0,C 180,E1 -23671.237,E2 -23671.237} C_VEL
LIN {X 0,Y 325.059,Z 451.269,A -85,B 0,C 180,E1 -23672.478,E2 -23672.478} C_VEL
LIN {X 0,Y 323.83,Z 450.831,A -85,B 0,C 180,E1 -23673.733,E2 -23673.733} C_VEL
LIN {X 0,Y 322.193,Z 450.145,A -85,B 0,C 180,E1 -23675.006,E2 -23675.006} C_VEL
LIN {X 0,Y 318.726,Z 448.398,A -85,B 0,C 180,E1 -23677.139,E2 -23677.139} C_VEL
LIN {X 0,Y 315.019,Z 446.181,A -85,B 0,C 180,E1 -23678.985,E2 -23678.985} C_VEL
LIN {X 0,Y 311.828,Z 443.98,A -85,B 0,C 180,E1 -23680.387,E2 -23680.387} C_VEL
LIN {X 0,Y 307.853,Z 441.292,A -85,B 0,C 180,E1 -23681.856,E2 -23681.856} C_VEL
LIN {X 0,Y 302.617,Z 438,A -85,B 0,C 180,E1 -23683.429,E2 -23683.429} C_VEL
LIN {X 0,Y 296.484,Z 433.751,A -85,B 0,C 180,E1 -23685.114,E2 -23685.114} C_VEL
LIN {X 0,Y 289.831,Z 429.117,A -85,B 0,C 180,E1 -23686.706,E2 -23686.706} C_VEL
LIN {X 0,Y 278.837,Z 421.693,A -85,B 0,C 180,E1 -23689.127,E2 -23689.127} C_VEL
LIN {X 0,Y 265.357,Z 412.539,A -85,B 0,C 180,E1 -23692.034,E2 -23692.034} C_VEL
LIN {X 0,Y 253.572,Z 403.678,A -85,B 0,C 180,E1 -23694.717,E2 -23694.717} C_VEL
LIN {X 0,Y 242.786,Z 394.274,A -85,B 0,C 180,E1 -23697.374,E2 -23697.374} C_VEL
LIN {X 0,Y 233.382,Z 384.466,A -85,B 0,C 180,E1 -23699.887,E2 -23699.887} C_VEL
LIN {X 0,Y 223.049,Z 372.001,A -85,B 0,C 180,E1 -23702.768,E2 -23702.768} C_VEL
LIN {X 0,Y 214.891,Z 360.738,A -85,B 0,C 180,E1 -23705.052,E2 -23705.052} C_VEL
LIN {X 0,Y 206.616,Z 347.706,A -85,B 0,C 180,E1 -23707.331,E2 -23707.331} C_VEL
LIN {X 0,Y 199.846,Z 334.967,A -85,B 0,C 180,E1 -23709.416,E2 -23709.416} C_VEL
LIN {X 0,Y 191.134,Z 315.423,A -85,B 0,C 180,E1 -23712.585,E2 -23712.585} C_VEL
LIN {X 0,Y 185.214,Z 303.601,A -85,B 0,C 180,E1 -23714.936,E2 -23714.936} C_VEL
LIN {X 0,Y 178.874,Z 292.837,A -85,B 0,C 180,E1 -23717.641,E2 -23717.641} C_VEL
LIN {X 0,Y 173.472,Z 284.657,A -85,B 0,C 180,E1 -23720.168,E2 -23720.168} C_VEL
LIN {X 0,Y 170.319,Z 280.225,A -85,B 0,C 180,E1 -23721.762,E2 -23721.762} C_VEL
LIN {X 0,Y 168.206,Z 277.214,A -85,B 0,C 180,E1 -23722.9,E2 -23722.9} C_VEL
LIN {X 0,Y 165.706,Z 273.887,A -85,B 0,C 180,E1 -23724.31,E2 -23724.31} C_VEL
LIN {X 0,Y 164.769,Z 272.694,A -85,B 0,C 180,E1 -23724.858,E2 -23724.858} C_VEL
LIN {X 0,Y 162.353,Z 269.892,A -85,B 0,C 180,E1 -23726.316,E2 -23726.316} C_VEL
LIN {X 0,Y 161.127,Z 267.829,A -85,B 0,C 180,E1 -23727.148,E2 -23727.148} C_VEL
LIN {X 0,Y 158.716,Z 265.785,A -85,B 0,C 180,E1 -23728.707,E2 -23728.707} C_VEL
LIN {X 0,Y 157.461,Z 263.121,A -85,B 0,C 180,E1 -23729.861,E2 -23729.861} C_VEL
LIN {X 0,Y 157.279,Z 262.435,A -85,B 0,C 180,E1 -23730.927,E2 -23730.927} C_VEL
LIN {X 0,Y 157.312,Z 262.351,A -85,B 0,C 180,E1 -23733.466,E2 -23733.466} C_VEL
LIN {X 0,Y 157.39,Z 262.335,A -85,B 0,C 180,E1 -23739.671,E2 -23739.671} C_VEL
LIN {X 0,Y 157.469,Z 262.359,A -85,B 0,C 180,E1 -23744.469,E2 -23744.469} C_VEL
LIN {X 0,Y 157.69,Z 262.287,A -85,B 0,C 180,E1 -23749.732,E2 -23749.732} C_VEL
LIN {X 0,Y 157.77,Z 262.292,A -85,B 0,C 180,E1 -23752.322,E2 -23752.322} C_VEL
LIN {X 0,Y 158.256,Z 262.214,A -85,B 0,C 180,E1 -23760.001,E2 -23760.001} C_VEL
LIN {X 0,Y 157.762,Z 262.286,A -85,B 0,C 180,E1 -23767.682,E2 -23767.682} C_VEL
LIN {X 0,Y 157.633,Z 262.3,A -85,B 0,C 180,E1 -23771.23,E2 -23771.23} C_VEL
LIN {X 0,Y 157.436,Z 262.35,A -85,B 0,C 180,E1 -23775.537,E2 -23775.537} C_VEL
LIN {X 0,Y 157.37,Z 262.345,A -85,B 0,C 180,E1 -23780.934,E2 -23780.934} C_VEL
LIN {X 0,Y 157.311,Z 262.347,A -85,B 0,C 180,E1 -23786.682,E2 -23786.682} C_VEL
LIN {X 0,Y 157.338,Z 262.677,A -85,B 0,C 180,E1 -23789.339,E2 -23789.339} C_VEL
LIN {X 0,Y 157.611,Z 263.709,A -85,B 0,C 180,E1 -23790.018,E2 -23790.018} C_VEL
LIN {X 0,Y 159.137,Z 266.277,A -85,B 0,C 180,E1 -23791.204,E2 -23791.204} C_VEL
LIN {X 0,Y 161.465,Z 268.181,A -85,B 0,C 180,E1 -23792.685,E2 -23792.685} C_VEL
LIN {X 0,Y 163.44,Z 271.403,A -85,B 0,C 180,E1 -23793.989,E2 -23793.989} C_VEL
LIN {X 0,Y 165.36,Z 273.333,A -85,B 0,C 180,E1 -23795.099,E2 -23795.099} C_VEL
LIN {X 0,Y 167.971,Z 277.084,A -85,B 0,C 180,E1 -23796.602,E2 -23796.602} C_VEL
LIN {X 0,Y 172.505,Z 284.488,A -85,B 0,C 180,E1 -23799.05,E2 -23799.05} C_VEL
LIN {X 0,Y 176.658,Z 291.926,A -85,B 0,C 180,E1 -23801.122,E2 -23801.122} C_VEL
LIN {X 0,Y 182.848,Z 304.28,A -85,B 0,C 180,E1 -23803.97,E2 -23803.97} C_VEL
LIN {X 0,Y 188.716,Z 318.658,A -85,B 0,C 180,E1 -23806.516,E2 -23806.516} C_VEL
LIN {X 0,Y 189.738,Z 322,A -85,B 0,C 180,E1 -23806.975,E2 -23806.975} C_VEL
LIN {X 0,Y 190.617,Z 329.588,A -85,B 0,C 180,E1 -23807.599,E2 -23807.599} C_VEL
LIN {X 0,Y 188.221,Z 367.873,A -85,B 0,C 180,E1 -23808.941,E2 -23808.941} C_VEL
LIN {X 0,Y 186.865,Z 379.112,A -85,B 0,C 180,E1 -23809.579,E2 -23809.579} C_VEL
LIN {X 0,Y 184.668,Z 391.333,A -85,B 0,C 180,E1 -23810.574,E2 -23810.574} C_VEL
LIN {X 0,Y 181.499,Z 404.042,A -85,B 0,C 180,E1 -23812.069,E2 -23812.069} C_VEL
LIN {X 0,Y 178.748,Z 413.313,A -85,B 0,C 180,E1 -23813.51,E2 -23813.51} C_VEL
LIN {X 0,Y 175.735,Z 422.254,A -85,B 0,C 180,E1 -23815.258,E2 -23815.258} C_VEL
LIN {X 0,Y 172.458,Z 430.777,A -85,B 0,C 180,E1 -23817.319,E2 -23817.319} C_VEL
LIN {X 0,Y 169.47,Z 437.993,A -85,B 0,C 180,E1 -23819.469,E2 -23819.469} C_VEL
LIN {X 0,Y 166.766,Z 444.193,A -85,B 0,C 180,E1 -23821.699,E2 -23821.699} C_VEL
LIN {X 0,Y 163.9,Z 450.733,A -85,B 0,C 180,E1 -23824.609,E2 -23824.609} C_VEL
LIN {X 0,Y 161.718,Z 455.233,A -85,B 0,C 180,E1 -23826.976,E2 -23826.976} C_VEL
LIN {X 0,Y 159.063,Z 460.725,A -85,B 0,C 180,E1 -23830.648,E2 -23830.648} C_VEL
LIN {X 0,Y 157.001,Z 465.052,A -85,B 0,C 180,E1 -23834.42,E2 -23834.42} C_VEL
LIN {X 0,Y 156.079,Z 467.424,A -85,B 0,C 180,E1 -23836.989,E2 -23836.989} C_VEL
LIN {X 0,Y 155.401,Z 469.229,A -85,B 0,C 180,E1 -23839.578,E2 -23839.578} C_VEL
LIN {X 0,Y 154.754,Z 471.687,A -85,B 0,C 180,E1 -23844.789,E2 -23844.789} C_VEL
LIN {X 0,Y 154.715,Z 472.403,A -85,B 0,C 180,E1 -23847.983,E2 -23847.983} C_VEL
LIN {X 0,Y 154.687,Z 472.433,A -85,B 0,C 180,E1 -23851.695,E2 -23851.695} C_VEL
LIN {X 0,Y 154.694,Z 471.686,A -85,B 0,C 180,E1 -23855.213,E2 -23855.213} C_VEL
LIN {X 0,Y 155.354,Z 469.227,A -85,B 0,C 180,E1 -23860.425,E2 -23860.425} C_VEL
LIN {X 0,Y 156.525,Z 466.272,A -85,B 0,C 180,E1 -23864.297,E2 -23864.297} C_VEL
LIN {X 0,Y 158.287,Z 462.279,A -85,B 0,C 180,E1 -23868.108,E2 -23868.108} C_VEL
LIN {X 0,Y 160.763,Z 457.148,A -85,B 0,C 180,E1 -23871.814,E2 -23871.814} C_VEL
LIN {X 0,Y 163.346,Z 451.889,A -85,B 0,C 180,E1 -23874.803,E2 -23874.803} C_VEL
LIN {X 0,Y 166.149,Z 445.569,A -85,B 0,C 180,E1 -23877.729,E2 -23877.729} C_VEL
LIN {X 0,Y 166.624,Z 444.506,A -85,B 0,C 180,E1 -23878.171,E2 -23878.171} C_VEL
LIN {X 0,Y 167.687,Z 440.818,A -85,B 0,C 180,E1 -23879.712,E2 -23879.712} C_VEL
LIN {X 0,Y 167.951,Z 434.408,A -85,B 0,C 180,E1 -23882.3,E2 -23882.3} C_VEL
LIN {X 0,Y 168.4,Z 427.519,A -85,B 0,C 180,E1 -23884.719,E2 -23884.719} C_VEL
LIN {X 0,Y 169.617,Z 422.928,A -85,B 0,C 180,E1 -23885.908,E2 -23885.908} C_VEL
LIN {X 0,Y 172.6,Z 414.47,A -85,B 0,C 180,E1 -23887.646,E2 -23887.646} C_VEL
LIN {X 0,Y 175.446,Z 405.479,A -85,B 0,C 180,E1 -23889.117,E2 -23889.117} C_VEL
LIN {X 0,Y 178.228,Z 395.346,A -85,B 0,C 180,E1 -23890.404,E2 -23890.404} C_VEL
LIN {X 0,Y 180.804,Z 383.291,A -85,B 0,C 180,E1 -23891.565,E2 -23891.565} C_VEL
LIN {X 0,Y 182.748,Z 369.966,A -85,B 0,C 180,E1 -23892.403,E2 -23892.403} C_VEL
LIN {X 0,Y 184.061,Z 351.75,A -85,B 0,C 180,E1 -23893.113,E2 -23893.113} C_VEL
LIN {X 0,Y 185.341,Z 329.452,A -85,B 0,C 180,E1 -23893.905,E2 -23893.905} C_VEL
LIN {X 0,Y 184.457,Z 323.48,A -85,B 0,C 180,E1 -23894.486,E2 -23894.486} C_VEL
LIN {X 0,Y 179.005,Z 309.648,A -85,B 0,C 180,E1 -23897.003,E2 -23897.003} C_VEL
LIN {X 0,Y 174.222,Z 299.533,A -85,B 0,C 180,E1 -23899.326,E2 -23899.326} C_VEL
LIN {X 0,Y 169.591,Z 290.719,A -85,B 0,C 180,E1 -23901.754,E2 -23901.754} C_VEL
LIN {X 0,Y 164.994,Z 282.878,A -85,B 0,C 180,E1 -23904.379,E2 -23904.379} C_VEL
LIN {X 0,Y 161.848,Z 278.572,A -85,B 0,C 180,E1 -23906.287,E2 -23906.287} C_VEL
LIN {X 0,Y 159.209,Z 275.128,A -85,B 0,C 180,E1 -23908.012,E2 -23908.012} C_VEL
LIN {X 0,Y 158.448,Z 274.008,A -85,B 0,C 180,E1 -23908.547,E2 -23908.547} C_VEL
LIN {X 0,Y 155.972,Z 271.452,A -85,B 0,C 180,E1 -23910.286,E2 -23910.286} C_VEL
LIN {X 0,Y 154.522,Z 268.932,A -85,B 0,C 180,E1 -23911.472,E2 -23911.472} C_VEL
LIN {X 0,Y 151.762,Z 266.786,A -85,B 0,C 180,E1 -23913.657,E2 -23913.657} C_VEL
LIN {X 0,Y 150.346,Z 263.925,A -85,B 0,C 180,E1 -23915.304,E2 -23915.304} C_VEL
LIN {X 0,Y 150.279,Z 263.297,A -85,B 0,C 180,E1 -23916.576,E2 -23916.576} C_VEL
LIN {X 0,Y 150.339,Z 263.205,A -85,B 0,C 180,E1 -23920.898,E2 -23920.898} C_VEL
LIN {X 0,Y 150.422,Z 263.234,A -85,B 0,C 180,E1 -23926.489,E2 -23926.489} C_VEL
LIN {X 0,Y 150.608,Z 263.17,A -85,B 0,C 180,E1 -23929.241,E2 -23929.241} C_VEL
LIN {X 0,Y 150.684,Z 263.163,A -85,B 0,C 180,E1 -23931.955,E2 -23931.955} C_VEL
LIN {X 0,Y 151.216,Z 263.09,A -85,B 0,C 180,E1 -23939.999,E2 -23939.999} C_VEL
LIN {X 0,Y 150.707,Z 263.166,A -85,B 0,C 180,E1 -23948.041,E2 -23948.041} C_VEL
LIN {X 0,Y 150.577,Z 263.178,A -85,B 0,C 180,E1 -23951.437,E2 -23951.437} C_VEL
LIN {X 0,Y 150.374,Z 263.226,A -85,B 0,C 180,E1 -23956.284,E2 -23956.284} C_VEL
LIN {X 0,Y 150.348,Z 263.215,A -85,B 0,C 180,E1 -23960.789,E2 -23960.789} C_VEL
LIN {X 0,Y 150.258,Z 263.5,A -85,B 0,C 180,E1 -23964.617,E2 -23964.617} C_VEL
LIN {X 0,Y 150.546,Z 264.611,A -85,B 0,C 180,E1 -23965.503,E2 -23965.503} C_VEL
LIN {X 0,Y 152.173,Z 267.257,A -85,B 0,C 180,E1 -23967.081,E2 -23967.081} C_VEL
LIN {X 0,Y 154.795,Z 269.197,A -85,B 0,C 180,E1 -23969.119,E2 -23969.119} C_VEL
LIN {X 0,Y 156.68,Z 272.391,A -85,B 0,C 180,E1 -23970.627,E2 -23970.627} C_VEL
LIN {X 0,Y 158.909,Z 274.543,A -85,B 0,C 180,E1 -23972.149,E2 -23972.149} C_VEL
LIN {X 0,Y 161.502,Z 278.233,A -85,B 0,C 180,E1 -23973.885,E2 -23973.885} C_VEL
LIN {X 0,Y 162.765,Z 279.665,A -85,B 0,C 180,E1 -23974.656,E2 -23974.656} C_VEL
LIN {X 0,Y 166.99,Z 285.596,A -85,B 0,C 180,E1 -23977.132,E2 -23977.132} C_VEL
LIN {X 0,Y 171.286,Z 291.838,A -85,B 0,C 180,E1 -23979.41,E2 -23979.41} C_VEL
LIN {X 0,Y 177.736,Z 302.283,A -85,B 0,C 180,E1 -23982.51,E2 -23982.51} C_VEL
LIN {X 0,Y 183.744,Z 313.411,A -85,B 0,C 180,E1 -23985.135,E2 -23985.135} C_VEL
LIN {X 0,Y 189.751,Z 326.695,A -85,B 0,C 180,E1 -23987.598,E2 -23987.598} C_VEL
LIN {X 0,Y 197.12,Z 343.245,A -85,B 0,C 180,E1 -23990.311,E2 -23990.311} C_VEL
LIN {X 0,Y 205.091,Z 357.526,A -85,B 0,C 180,E1 -23992.816,E2 -23992.816} C_VEL
LIN {X 0,Y 211.511,Z 367.66,A -85,B 0,C 180,E1 -23994.802,E2 -23994.802} C_VEL
LIN {X 0,Y 218.163,Z 376.993,A -85,B 0,C 180,E1 -23996.883,E2 -23996.883} C_VEL
LIN {X 0,Y 226.031,Z 386.796,A -85,B 0,C 180,E1 -23999.303,E2 -23999.303} C_VEL
LIN {X 0,Y 234.953,Z 396.524,A -85,B 0,C 180,E1 -24001.933,E2 -24001.933} C_VEL
LIN {X 0,Y 246.243,Z 406.749,A -85,B 0,C 180,E1 -24004.979,E2 -24004.979} C_VEL
LIN {X 0,Y 257.983,Z 415.616,A -85,B 0,C 180,E1 -24007.852,E2 -24007.852} C_VEL
LIN {X 0,Y 271.467,Z 424.494,A -85,B 0,C 180,E1 -24010.897,E2 -24010.897} C_VEL
LIN {X 0,Y 279.632,Z 429.761,A -85,B 0,C 180,E1 -24012.753,E2 -24012.753} C_VEL
LIN {X 0,Y 287.859,Z 435.024,A -85,B 0,C 180,E1 -24014.656,E2 -24014.656} C_VEL
LIN {X 0,Y 293.567,Z 438.987,A -85,B 0,C 180,E1 -24016.149,E2 -24016.149} C_VEL
LIN {X 0,Y 299.407,Z 442.852,A -85,B 0,C 180,E1 -24017.804,E2 -24017.804} C_VEL
LIN {X 0,Y 304.163,Z 445.81,A -85,B 0,C 180,E1 -24019.348,E2 -24019.348} C_VEL
LIN {X 0,Y 307.594,Z 448.268,A -85,B 0,C 180,E1 -24020.797,E2 -24020.797} C_VEL
LIN {X 0,Y 311.708,Z 450.832,A -85,B 0,C 180,E1 -24022.767,E2 -24022.767} C_VEL
LIN {X 0,Y 315.29,Z 452.757,A -85,B 0,C 180,E1 -24024.885,E2 -24024.885} C_VEL
LIN {X 0,Y 317.053,Z 453.5,A -85,B 0,C 180,E1 -24026.187,E2 -24026.187} C_VEL
LIN {X 0,Y 318.367,Z 454.001,A -85,B 0,C 180,E1 -24027.47,E2 -24027.47} C_VEL
LIN {X 0,Y 319.072,Z 454.324,A -85,B 0,C 180,E1 -24028.738,E2 -24028.738} C_VEL
LIN {X 0,Y 319.442,Z 454.38,A -85,B 0,C 180,E1 -24030,E2 -24030} C_VEL
LIN {X 0,Y 319.087,Z 454.315,A -85,B 0,C 180,E1 -24031.262,E2 -24031.262} C_VEL
LIN {X 0,Y 318.39,Z 453.99,A -85,B 0,C 180,E1 -24032.53,E2 -24032.53} C_VEL
LIN {X 0,Y 316.981,Z 453.471,A -85,B 0,C 180,E1 -24033.878,E2 -24033.878} C_VEL
LIN {X 0,Y 315.286,Z 452.76,A -85,B 0,C 180,E1 -24035.115,E2 -24035.115} C_VEL
LIN {X 0,Y 311.699,Z 450.845,A -85,B 0,C 180,E1 -24037.22,E2 -24037.22} C_VEL
LIN {X 0,Y 307.591,Z 448.251,A -85,B 0,C 180,E1 -24039.203,E2 -24039.203} C_VEL
LIN {X 0,Y 304.111,Z 445.808,A -85,B 0,C 180,E1 -24040.654,E2 -24040.654} C_VEL
LIN {X 0,Y 298.219,Z 442.142,A -85,B 0,C 180,E1 -24042.543,E2 -24042.543} C_VEL
LIN {X 0,Y 290.565,Z 436.89,A -85,B 0,C 180,E1 -24044.652,E2 -24044.652} C_VEL
LIN {X 0,Y 282.37,Z 431.536,A -85,B 0,C 180,E1 -24046.62,E2 -24046.62} C_VEL
LIN {X 0,Y 271.453,Z 424.539,A -85,B 0,C 180,E1 -24049.095,E2 -24049.095} C_VEL
LIN {X 0,Y 257.992,Z 415.587,A -85,B 0,C 180,E1 -24052.153,E2 -24052.153} C_VEL
LIN {X 0,Y 246.245,Z 406.742,A -85,B 0,C 180,E1 -24055.022,E2 -24055.022} C_VEL
LIN {X 0,Y 236.178,Z 397.778,A -85,B 0,C 180,E1 -24057.717,E2 -24057.717} C_VEL
LIN {X 0,Y 226.044,Z 386.845,A -85,B 0,C 180,E1 -24060.688,E2 -24060.688} C_VEL
LIN {X 0,Y 217.124,Z 375.531,A -85,B 0,C 180,E1 -24063.458,E2 -24063.458} C_VEL
LIN {X 0,Y 209.767,Z 364.945,A -85,B 0,C 180,E1 -24065.767,E2 -24065.767} C_VEL
LIN {X 0,Y 202.081,Z 352.412,A -85,B 0,C 180,E1 -24068.116,E2 -24068.116} C_VEL
LIN {X 0,Y 195.278,Z 339.462,A -85,B 0,C 180,E1 -24070.321,E2 -24070.321} C_VEL
LIN {X 0,Y 186.646,Z 319.612,A -85,B 0,C 180,E1 -24073.654,E2 -24073.654} C_VEL
LIN {X 0,Y 180.961,Z 308.042,A -85,B 0,C 180,E1 -24076.055,E2 -24076.055} C_VEL
LIN {X 0,Y 174.974,Z 297.703,A -85,B 0,C 180,E1 -24078.772,E2 -24078.772} C_VEL
LIN {X 0,Y 168.362,Z 287.4,A -85,B 0,C 180,E1 -24082.128,E2 -24082.128} C_VEL
LIN {X 0,Y 164.906,Z 282.693,A -85,B 0,C 180,E1 -24084.053,E2 -24084.053} C_VEL
LIN {X 0,Y 162.06,Z 278.768,A -85,B 0,C 180,E1 -24085.779,E2 -24085.779} C_VEL
LIN {X 0,Y 159.404,Z 275.44,A -85,B 0,C 180,E1 -24087.493,E2 -24087.493} C_VEL
LIN {X 0,Y 158.411,Z 273.979,A -85,B 0,C 180,E1 -24088.189,E2 -24088.189} C_VEL
LIN {X 0,Y 155.942,Z 271.404,A -85,B 0,C 180,E1 -24089.927,E2 -24089.927} C_VEL
LIN {X 0,Y 154.503,Z 268.956,A -85,B 0,C 180,E1 -24091.1,E2 -24091.1} C_VEL
LIN {X 0,Y 151.774,Z 266.797,A -85,B 0,C 180,E1 -24093.265,E2 -24093.265} C_VEL
LIN {X 0,Y 150.365,Z 264.001,A -85,B 0,C 180,E1 -24094.861,E2 -24094.861} C_VEL
LIN {X 0,Y 150.256,Z 263.302,A -85,B 0,C 180,E1 -24096.209,E2 -24096.209} C_VEL
LIN {X 0,Y 150.364,Z 263.205,A -85,B 0,C 180,E1 -24100.904,E2 -24100.904} C_VEL
LIN {X 0,Y 150.443,Z 263.225,A -85,B 0,C 180,E1 -24106.494,E2 -24106.494} C_VEL
LIN {X 0,Y 150.611,Z 263.17,A -85,B 0,C 180,E1 -24109.244,E2 -24109.244} C_VEL
LIN {X 0,Y 150.707,Z 263.166,A -85,B 0,C 180,E1 -24111.959,E2 -24111.959} C_VEL
LIN {X 0,Y 151.216,Z 263.09,A -85,B 0,C 180,E1 -24120.001,E2 -24120.001} C_VEL
LIN {X 0,Y 150.684,Z 263.163,A -85,B 0,C 180,E1 -24128.045,E2 -24128.045} C_VEL
LIN {X 0,Y 150.575,Z 263.18,A -85,B 0,C 180,E1 -24131.432,E2 -24131.432} C_VEL
LIN {X 0,Y 150.348,Z 263.219,A -85,B 0,C 180,E1 -24136.29,E2 -24136.29} C_VEL
LIN {X 0,Y 150.352,Z 263.216,A -85,B 0,C 180,E1 -24140.793,E2 -24140.793} C_VEL
LIN {X 0,Y 150.279,Z 263.53,A -85,B 0,C 180,E1 -24144.248,E2 -24144.248} C_VEL
LIN {X 0,Y 150.587,Z 264.7,A -85,B 0,C 180,E1 -24145.168,E2 -24145.168} C_VEL
LIN {X 0,Y 152.139,Z 267.21,A -85,B 0,C 180,E1 -24146.669,E2 -24146.669} C_VEL
LIN {X 0,Y 154.802,Z 269.278,A -85,B 0,C 180,E1 -24148.749,E2 -24148.749} C_VEL
LIN {X 0,Y 156.711,Z 272.431,A -85,B 0,C 180,E1 -24150.268,E2 -24150.268} C_VEL
LIN {X 0,Y 158.932,Z 274.616,A -85,B 0,C 180,E1 -24151.786,E2 -24151.786} C_VEL
LIN {X 0,Y 161.516,Z 278.238,A -85,B 0,C 180,E1 -24153.511,E2 -24153.511} C_VEL
LIN {X 0,Y 162.827,Z 279.84,A -85,B 0,C 180,E1 -24154.319,E2 -24154.319} C_VEL
LIN {X 0,Y 165.768,Z 284.167,A -85,B 0,C 180,E1 -24156.082,E2 -24156.082} C_VEL
LIN {X 0,Y 170.881,Z 292.927,A -85,B 0,C 180,E1 -24158.933,E2 -24158.933} C_VEL
LIN {X 0,Y 177.936,Z 307.138,A -85,B 0,C 180,E1 -24162.483,E2 -24162.483} C_VEL
LIN {X 0,Y 183.554,Z 320.963,A -85,B 0,C 180,E1 -24165.103,E2 -24165.103} C_VEL
LIN {X 0,Y 184.742,Z 324.748,A -85,B 0,C 180,E1 -24165.668,E2 -24165.668} C_VEL
LIN {X 0,Y 185.38,Z 330.483,A -85,B 0,C 180,E1 -24166.16,E2 -24166.16} C_VEL
LIN {X 0,Y 182.938,Z 367.754,A -85,B 0,C 180,E1 -24167.489,E2 -24167.489} C_VEL
LIN {X 0,Y 181.399,Z 379.868,A -85,B 0,C 180,E1 -24168.193,E2 -24168.193} C_VEL
LIN {X 0,Y 178.725,Z 393.332,A -85,B 0,C 180,E1 -24169.362,E2 -24169.362} C_VEL
LIN {X 0,Y 175.955,Z 403.849,A -85,B 0,C 180,E1 -24170.649,E2 -24170.649} C_VEL
LIN {X 0,Y 173.087,Z 413.12,A -85,B 0,C 180,E1 -24172.111,E2 -24172.111} C_VEL
LIN {X 0,Y 169.95,Z 422.062,A -85,B 0,C 180,E1 -24173.894,E2 -24173.894} C_VEL
LIN {X 0,Y 166.52,Z 430.585,A -85,B 0,C 180,E1 -24175.998,E2 -24175.998} C_VEL
LIN {X 0,Y 163.368,Z 437.799,A -85,B 0,C 180,E1 -24178.198,E2 -24178.198} C_VEL
LIN {X 0,Y 160.517,Z 443.999,A -85,B 0,C 180,E1 -24180.491,E2 -24180.491} C_VEL
LIN {X 0,Y 157.472,Z 450.539,A -85,B 0,C 180,E1 -24183.494,E2 -24183.494} C_VEL
LIN {X 0,Y 155.2,Z 455.04,A -85,B 0,C 180,E1 -24185.949,E2 -24185.949} C_VEL
LIN {X 0,Y 152.354,Z 460.531,A -85,B 0,C 180,E1 -24189.759,E2 -24189.759} C_VEL
LIN {X 0,Y 150.133,Z 464.858,A -85,B 0,C 180,E1 -24193.688,E2 -24193.688} C_VEL
LIN {X 0,Y 149.134,Z 467.23,A -85,B 0,C 180,E1 -24196.372,E2 -24196.372} C_VEL
LIN {X 0,Y 148.387,Z 469.035,A -85,B 0,C 180,E1 -24199.079,E2 -24199.079} C_VEL
LIN {X 0,Y 147.686,Z 471.495,A -85,B 0,C 180,E1 -24204.539,E2 -24204.539} C_VEL
LIN {X 0,Y 147.628,Z 472.246,A -85,B 0,C 180,E1 -24208.73,E2 -24208.73} C_VEL
LIN {X 0,Y 147.571,Z 472.088,A -85,B 0,C 180,E1 -24212.73,E2 -24212.73} C_VEL
LIN {X 0,Y 147.621,Z 471.493,A -85,B 0,C 180,E1 -24215.464,E2 -24215.464} C_VEL
LIN {X 0,Y 148.351,Z 469.034,A -85,B 0,C 180,E1 -24220.923,E2 -24220.923} C_VEL
LIN {X 0,Y 149.625,Z 466.078,A -85,B 0,C 180,E1 -24224.972,E2 -24224.972} C_VEL
LIN {X 0,Y 151.542,Z 462.086,A -85,B 0,C 180,E1 -24228.943,E2 -24228.943} C_VEL
LIN {X 0,Y 154.152,Z 456.954,A -85,B 0,C 180,E1 -24232.801,E2 -24232.801} C_VEL
LIN {X 0,Y 156.902,Z 451.695,A -85,B 0,C 180,E1 -24235.895,E2 -24235.895} C_VEL
LIN {X 0,Y 159.083,Z 447.108,A -85,B 0,C 180,E1 -24238.168,E2 -24238.168} C_VEL
LIN {X 0,Y 161.902,Z 441.052,A -85,B 0,C 180,E1 -24240.667,E2 -24240.667} C_VEL
LIN {X 0,Y 165.741,Z 432.504,A -85,B 0,C 180,E1 -24243.452,E2 -24243.452} C_VEL
LIN {X 0,Y 169.052,Z 424.329,A -85,B 0,C 180,E1 -24245.593,E2 -24245.593} C_VEL
LIN {X 0,Y 169.617,Z 422.928,A -85,B 0,C 180,E1 -24245.908,E2 -24245.908} C_VEL
LIN {X 0,Y 170.249,Z 419.875,A -85,B 0,C 180,E1 -24246.734,E2 -24246.734} C_VEL
LIN {X 0,Y 169.081,Z 409.896,A -85,B 0,C 180,E1 -24249.793,E2 -24249.793} C_VEL
LIN {X 0,Y 169.643,Z 406.426,A -85,B 0,C 180,E1 -24250.457,E2 -24250.457} C_VEL
LIN {X 0,Y 172.374,Z 397.166,A -85,B 0,C 180,E1 -24251.689,E2 -24251.689} C_VEL
LIN {X 0,Y 174.452,Z 388.375,A -85,B 0,C 180,E1 -24252.634,E2 -24252.634} C_VEL
LIN {X 0,Y 176.382,Z 378.34,A -85,B 0,C 180,E1 -24253.432,E2 -24253.432} C_VEL
LIN {X 0,Y 177.732,Z 368.218,A -85,B 0,C 180,E1 -24254.013,E2 -24254.013} C_VEL
LIN {X 0,Y 179.725,Z 339.89,A -85,B 0,C 180,E1 -24255.063,E2 -24255.063} C_VEL
LIN {X 0,Y 180.226,Z 330.607,A -85,B 0,C 180,E1 -24255.417,E2 -24255.417} C_VEL
LIN {X 0,Y 179.581,Z 326.369,A -85,B 0,C 180,E1 -24255.862,E2 -24255.862} C_VEL
LIN {X 0,Y 174.303,Z 312.753,A -85,B 0,C 180,E1 -24258.487,E2 -24258.487} C_VEL
LIN {X 0,Y 169.128,Z 301.693,A -85,B 0,C 180,E1 -24261.22,E2 -24261.22} C_VEL
LIN {X 0,Y 164.555,Z 292.969,A -85,B 0,C 180,E1 -24263.858,E2 -24263.858} C_VEL
LIN {X 0,Y 161.466,Z 287.871,A -85,B 0,C 180,E1 -24265.766,E2 -24265.766} C_VEL
LIN {X 0,Y 158.879,Z 284.274,A -85,B 0,C 180,E1 -24267.446,E2 -24267.446} C_VEL
LIN {X 0,Y 155.699,Z 279.968,A -85,B 0,C 180,E1 -24269.694,E2 -24269.694} C_VEL
LIN {X 0,Y 153.14,Z 276.857,A -85,B 0,C 180,E1 -24271.658,E2 -24271.658} C_VEL
LIN {X 0,Y 152.17,Z 275.306,A -85,B 0,C 180,E1 -24272.492,E2 -24272.492} C_VEL
LIN {X 0,Y 149.567,Z 272.923,A -85,B 0,C 180,E1 -24274.715,E2 -24274.715} C_VEL
LIN {X 0,Y 147.811,Z 269.959,A -85,B 0,C 180,E1 -24276.532,E2 -24276.532} C_VEL
LIN {X 0,Y 145.296,Z 268.214,A -85,B 0,C 180,E1 -24279.143,E2 -24279.143} C_VEL
LIN {X 0,Y 143.643,Z 265.628,A -85,B 0,C 180,E1 -24281.362,E2 -24281.362} C_VEL
LIN {X 0,Y 143.314,Z 264.414,A -85,B 0,C 180,E1 -24282.703,E2 -24282.703} C_VEL
LIN {X 0,Y 143.501,Z 264.062,A -85,B 0,C 180,E1 -24288.379,E2 -24288.379} C_VEL
LIN {X 0,Y 143.61,Z 264.04,A -85,B 0,C 180,E1 -24291.556,E2 -24291.556} C_VEL
LIN {X 0,Y 144.175,Z 263.966,A -85,B 0,C 180,E1 -24299.998,E2 -24299.998} C_VEL
LIN {X 0,Y 143.628,Z 264.043,A -85,B 0,C 180,E1 -24308.44,E2 -24308.44} C_VEL
LIN {X 0,Y 143.506,Z 264.06,A -85,B 0,C 180,E1 -24311.631,E2 -24311.631} C_VEL
LIN {X 0,Y 143.34,Z 264.381,A -85,B 0,C 180,E1 -24317.659,E2 -24317.659} C_VEL
LIN {X 0,Y 143.652,Z 265.511,A -85,B 0,C 180,E1 -24319.003,E2 -24319.003} C_VEL
LIN {X 0,Y 145.175,Z 268.119,A -85,B 0,C 180,E1 -24321.102,E2 -24321.102} C_VEL
LIN {X 0,Y 147.799,Z 269.949,A -85,B 0,C 180,E1 -24323.838,E2 -24323.838} C_VEL
LIN {X 0,Y 150.304,Z 273.826,A -85,B 0,C 180,E1 -24326.347,E2 -24326.347} C_VEL
LIN {X 0,Y 152.611,Z 275.856,A -85,B 0,C 180,E1 -24328.258,E2 -24328.258} C_VEL
LIN {X 0,Y 154.788,Z 279.118,A -85,B 0,C 180,E1 -24330.033,E2 -24330.033} C_VEL
LIN {X 0,Y 156.561,Z 281.046,A -85,B 0,C 180,E1 -24331.313,E2 -24331.313} C_VEL
LIN {X 0,Y 159.489,Z 284.913,A -85,B 0,C 180,E1 -24333.327,E2 -24333.327} C_VEL
LIN {X 0,Y 164.483,Z 292.041,A -85,B 0,C 180,E1 -24336.423,E2 -24336.423} C_VEL
LIN {X 0,Y 169.947,Z 300.536,A -85,B 0,C 180,E1 -24339.427,E2 -24339.427} C_VEL
LIN {X 0,Y 175.372,Z 309.904,A -85,B 0,C 180,E1 -24342.114,E2 -24342.114} C_VEL
LIN {X 0,Y 180.271,Z 319.505,A -85,B 0,C 180,E1 -24344.361,E2 -24344.361} C_VEL
LIN {X 0,Y 185.631,Z 331.831,A -85,B 0,C 180,E1 -24346.686,E2 -24346.686} C_VEL
LIN {X 0,Y 192.273,Z 347.112,A -85,B 0,C 180,E1 -24349.281,E2 -24349.281} C_VEL
LIN {X 0,Y 200.018,Z 361.496,A -85,B 0,C 180,E1 -24351.931,E2 -24351.931} C_VEL
LIN {X 0,Y 207.275,Z 373.376,A -85,B 0,C 180,E1 -24354.463,E2 -24354.463} C_VEL
LIN {X 0,Y 215.796,Z 385.309,A -85,B 0,C 180,E1 -24357.428,E2 -24357.428} C_VEL
LIN {X 0,Y 224.478,Z 395.701,A -85,B 0,C 180,E1 -24360.317,E2 -24360.317} C_VEL
LIN {X 0,Y 232.853,Z 404.322,A -85,B 0,C 180,E1 -24362.919,E2 -24362.919} C_VEL
LIN {X 0,Y 242.851,Z 412.827,A -85,B 0,C 180,E1 -24365.728,E2 -24365.728} C_VEL
LIN {X 0,Y 255.915,Z 422.063,A -85,B 0,C 180,E1 -24369.019,E2 -24369.019} C_VEL
LIN {X 0,Y 269.436,Z 430.456,A -85,B 0,C 180,E1 -24372.183,E2 -24372.183} C_VEL
LIN {X 0,Y 280.405,Z 437.104,A -85,B 0,C 180,E1 -24374.783,E2 -24374.783} C_VEL
LIN {X 0,Y 288.574,Z 442.409,A -85,B 0,C 180,E1 -24376.945,E2 -24376.945} C_VEL
LIN {X 0,Y 294.028,Z 445.899,A -85,B 0,C 180,E1 -24378.517,E2 -24378.517} C_VEL
LIN {X 0,Y 298.023,Z 448.438,A -85,B 0,C 180,E1 -24379.813,E2 -24379.813} C_VEL
LIN {X 0,Y 302.985,Z 451.865,A -85,B 0,C 180,E1 -24382,E2 -24382} C_VEL
LIN {X 0,Y 305.818,Z 453.54,A -85,B 0,C 180,E1 -24383.402,E2 -24383.402} C_VEL
LIN {X 0,Y 308.113,Z 454.768,A -85,B 0,C 180,E1 -24384.765,E2 -24384.765} C_VEL
LIN {X 0,Y 310.054,Z 455.67,A -85,B 0,C 180,E1 -24386.101,E2 -24386.101} C_VEL
LIN {X 0,Y 311.475,Z 456.23,A -85,B 0,C 180,E1 -24387.414,E2 -24387.414} C_VEL
LIN {X 0,Y 312.293,Z 456.562,A -85,B 0,C 180,E1 -24388.71,E2 -24388.71} C_VEL
LIN {X 0,Y 312.711,Z 456.629,A -85,B 0,C 180,E1 -24390,E2 -24390} C_VEL
LIN {X 0,Y 312.308,Z 456.56,A -85,B 0,C 180,E1 -24391.289,E2 -24391.289} C_VEL
LIN {X 0,Y 311.508,Z 456.224,A -85,B 0,C 180,E1 -24392.586,E2 -24392.586} C_VEL
LIN {X 0,Y 309.97,Z 455.643,A -85,B 0,C 180,E1 -24393.966,E2 -24393.966} C_VEL
LIN {X 0,Y 308.114,Z 454.787,A -85,B 0,C 180,E1 -24395.235,E2 -24395.235} C_VEL
LIN {X 0,Y 304.615,Z 452.848,A -85,B 0,C 180,E1 -24397.221,E2 -24397.221} C_VEL
LIN {X 0,Y 299.759,Z 449.66,A -85,B 0,C 180,E1 -24399.446,E2 -24399.446} C_VEL
LIN {X 0,Y 297.996,Z 448.44,A -85,B 0,C 180,E1 -24400.187,E2 -24400.187} C_VEL
LIN {X 0,Y 294.032,Z 445.896,A -85,B 0,C 180,E1 -24401.486,E2 -24401.486} C_VEL
LIN {X 0,Y 285.855,Z 440.614,A -85,B 0,C 180,E1 -24403.805,E2 -24403.805} C_VEL
LIN {X 0,Y 277.642,Z 435.496,A -85,B 0,C 180,E1 -24405.87,E2 -24405.87} C_VEL
LIN {X 0,Y 266.696,Z 428.857,A -85,B 0,C 180,E1 -24408.44,E2 -24408.44} C_VEL
LIN {X 0,Y 252.311,Z 419.722,A -85,B 0,C 180,E1 -24411.843,E2 -24411.843} C_VEL
LIN {X 0,Y 239.053,Z 409.797,A -85,B 0,C 180,E1 -24415.31,E2 -24415.31} C_VEL
LIN {X 0,Y 228.035,Z 399.624,A -85,B 0,C 180,E1 -24418.541,E2 -24418.541} C_VEL
LIN {X 0,Y 219.809,Z 390.339,A -85,B 0,C 180,E1 -24421.211,E2 -24421.211} C_VEL
LIN {X 0,Y 211.795,Z 379.871,A -85,B 0,C 180,E1 -24423.947,E2 -24423.947} C_VEL
LIN {X 0,Y 205.416,Z 370.478,A -85,B 0,C 180,E1 -24426.176,E2 -24426.176} C_VEL
LIN {X 0,Y 198.596,Z 358.971,A -85,B 0,C 180,E1 -24428.57,E2 -24428.57} C_VEL
LIN {X 0,Y 191.253,Z 344.985,A -85,B 0,C 180,E1 -24431.088,E2 -24431.088} C_VEL
LIN {X 0,Y 181.936,Z 323.209,A -85,B 0,C 180,E1 -24434.899,E2 -24434.899} C_VEL
LIN {X 0,Y 176.689,Z 312.311,A -85,B 0,C 180,E1 -24437.27,E2 -24437.27} C_VEL
LIN {X 0,Y 171.193,Z 302.592,A -85,B 0,C 180,E1 -24439.934,E2 -24439.934} C_VEL
LIN {X 0,Y 165.165,Z 292.939,A -85,B 0,C 180,E1 -24443.191,E2 -24443.191} C_VEL
LIN {X 0,Y 161.183,Z 287.418,A -85,B 0,C 180,E1 -24445.567,E2 -24445.567} C_VEL
LIN {X 0,Y 158.95,Z 284.337,A -85,B 0,C 180,E1 -24447.018,E2 -24447.018} C_VEL
LIN {X 0,Y 155.815,Z 280.107,A -85,B 0,C 180,E1 -24449.227,E2 -24449.227} C_VEL
LIN {X 0,Y 153.217,Z 277.005,A -85,B 0,C 180,E1 -24451.21,E2 -24451.21} C_VEL
LIN {X 0,Y 152.345,Z 275.458,A -85,B 0,C 180,E1 -24451.969,E2 -24451.969} C_VEL
LIN {X 0,Y 149.579,Z 272.952,A -85,B 0,C 180,E1 -24454.32,E2 -24454.32} C_VEL
LIN {X 0,Y 147.797,Z 269.968,A -85,B 0,C 180,E1 -24456.161,E2 -24456.161} C_VEL
LIN {X 0,Y 145.175,Z 268.119,A -85,B 0,C 180,E1 -24458.898,E2 -24458.898} C_VEL
LIN {X 0,Y 143.654,Z 265.496,A -85,B 0,C 180,E1 -24460.997,E2 -24460.997} C_VEL
LIN {X 0,Y 143.334,Z 264.396,A -85,B 0,C 180,E1 -24462.34,E2 -24462.34} C_VEL
LIN {X 0,Y 143.506,Z 264.06,A -85,B 0,C 180,E1 -24468.369,E2 -24468.369} C_VEL
LIN {X 0,Y 143.628,Z 264.043,A -85,B 0,C 180,E1 -24471.56,E2 -24471.56} C_VEL
LIN {X 0,Y 144.175,Z 263.966,A -85,B 0,C 180,E1 -24480.002,E2 -24480.002} C_VEL
LIN {X 0,Y 143.61,Z 264.04,A -85,B 0,C 180,E1 -24488.444,E2 -24488.444} C_VEL
LIN {X 0,Y 143.501,Z 264.062,A -85,B 0,C 180,E1 -24491.621,E2 -24491.621} C_VEL
LIN {X 0,Y 143.304,Z 264.407,A -85,B 0,C 180,E1 -24497.298,E2 -24497.298} C_VEL
LIN {X 0,Y 143.644,Z 265.627,A -85,B 0,C 180,E1 -24498.637,E2 -24498.637} C_VEL
LIN {X 0,Y 145.296,Z 268.214,A -85,B 0,C 180,E1 -24500.857,E2 -24500.857} C_VEL
LIN {X 0,Y 148.125,Z 270.322,A -85,B 0,C 180,E1 -24503.786,E2 -24503.786} C_VEL
LIN {X 0,Y 149.805,Z 273.224,A -85,B 0,C 180,E1 -24505.509,E2 -24505.509} C_VEL
LIN {X 0,Y 152.619,Z 275.901,A -85,B 0,C 180,E1 -24507.886,E2 -24507.886} C_VEL
LIN {X 0,Y 154.924,Z 279.227,A -85,B 0,C 180,E1 -24509.749,E2 -24509.749} C_VEL
LIN {X 0,Y 156.497,Z 280.948,A -85,B 0,C 180,E1 -24510.884,E2 -24510.884} C_VEL
LIN {X 0,Y 159.254,Z 284.677,A -85,B 0,C 180,E1 -24512.797,E2 -24512.797} C_VEL
LIN {X 0,Y 162.732,Z 289.888,A -85,B 0,C 180,E1 -24515.03,E2 -24515.03} C_VEL
LIN {X 0,Y 167.269,Z 297.94,A -85,B 0,C 180,E1 -24517.73,E2 -24517.73} C_VEL
LIN {X 0,Y 173.466,Z 310.79,A -85,B 0,C 180,E1 -24521.081,E2 -24521.081} C_VEL
LIN {X 0,Y 178.532,Z 323.428,A -85,B 0,C 180,E1 -24523.625,E2 -24523.625} C_VEL
LIN {X 0,Y 179.892,Z 327.742,A -85,B 0,C 180,E1 -24524.316,E2 -24524.316} C_VEL
LIN {X 0,Y 180.195,Z 332.109,A -85,B 0,C 180,E1 -24524.656,E2 -24524.656} C_VEL
LIN {X 0,Y 177.699,Z 368.246,A -85,B 0,C 180,E1 -24525.973,E2 -24525.973} C_VEL
LIN {X 0,Y 175.981,Z 380.998,A -85,B 0,C 180,E1 -24526.744,E2 -24526.744} C_VEL
LIN {X 0,Y 173.134,Z 394.146,A -85,B 0,C 180,E1 -24527.95,E2 -24527.95} C_VEL
LIN {X 0,Y 170.535,Z 403.656,A -85,B 0,C 180,E1 -24529.139,E2 -24529.139} C_VEL
LIN {X 0,Y 167.544,Z 412.928,A -85,B 0,C 180,E1 -24530.621,E2 -24530.621} C_VEL
LIN {X 0,Y 164.266,Z 421.869,A -85,B 0,C 180,E1 -24532.434,E2 -24532.434} C_VEL
LIN {X 0,Y 160.685,Z 430.392,A -85,B 0,C 180,E1 -24534.583,E2 -24534.583} C_VEL
LIN {X 0,Y 157.362,Z 437.606,A -85,B 0,C 180,E1 -24536.832,E2 -24536.832} C_VEL
LIN {X 0,Y 154.365,Z 443.806,A -85,B 0,C 180,E1 -24539.19,E2 -24539.19} C_VEL
LIN {X 0,Y 151.11,Z 450.345,A -85,B 0,C 180,E1 -24542.284,E2 -24542.284} C_VEL
LIN {X 0,Y 148.741,Z 454.847,A -85,B 0,C 180,E1 -24544.834,E2 -24544.834} C_VEL
LIN {X 0,Y 145.688,Z 460.338,A -85,B 0,C 180,E1 -24548.789,E2 -24548.789} C_VEL
LIN {X 0,Y 143.298,Z 464.664,A -85,B 0,C 180,E1 -24552.886,E2 -24552.886} C_VEL
LIN {X 0,Y 142.218,Z 467.037,A -85,B 0,C 180,E1 -24555.695,E2 -24555.695} C_VEL
LIN {X 0,Y 141.398,Z 468.842,A -85,B 0,C 180,E1 -24558.532,E2 -24558.532} C_VEL
LIN {X 0,Y 140.617,Z 471.302,A -85,B 0,C 180,E1 -24564.263,E2 -24564.263} C_VEL
LIN {X 0,Y 140.572,Z 472.055,A -85,B 0,C 180,E1 -24569.356,E2 -24569.356} C_VEL
LIN {X 0,Y 140.489,Z 471.896,A -85,B 0,C 180,E1 -24572.867,E2 -24572.867} C_VEL
LIN {X 0,Y 140.545,Z 471.3,A -85,B 0,C 180,E1 -24575.74,E2 -24575.74} C_VEL
LIN {X 0,Y 141.369,Z 468.841,A -85,B 0,C 180,E1 -24581.47,E2 -24581.47} C_VEL
LIN {X 0,Y 142.727,Z 465.884,A -85,B 0,C 180,E1 -24585.713,E2 -24585.713} C_VEL
LIN {X 0,Y 144.806,Z 461.892,A -85,B 0,C 180,E1 -24589.861,E2 -24589.861} C_VEL
LIN {X 0,Y 147.602,Z 456.761,A -85,B 0,C 180,E1 -24593.874,E2 -24593.874} C_VEL
LIN {X 0,Y 150.518,Z 451.501,A -85,B 0,C 180,E1 -24597.081,E2 -24597.081} C_VEL
LIN {X 0,Y 153.651,Z 445.181,A -85,B 0,C 180,E1 -24600.208,E2 -24600.208} C_VEL
LIN {X 0,Y 156.584,Z 439.232,A -85,B 0,C 180,E1 -24602.588,E2 -24602.588} C_VEL
LIN {X 0,Y 159.836,Z 432.31,A -85,B 0,C 180,E1 -24604.862,E2 -24604.862} C_VEL
LIN {X 0,Y 163.321,Z 424.136,A -85,B 0,C 180,E1 -24607.045,E2 -24607.045} C_VEL
LIN {X 0,Y 166.569,Z 415.629,A -85,B 0,C 180,E1 -24608.874,E2 -24608.874} C_VEL
LIN {X 0,Y 169.643,Z 406.426,A -85,B 0,C 180,E1 -24610.457,E2 -24610.457} C_VEL
LIN {X 0,Y 170.839,Z 401.26,A -85,B 0,C 180,E1 -24611.332,E2 -24611.332} C_VEL
LIN {X 0,Y 170.976,Z 392.641,A -85,B 0,C 180,E1 -24612.987,E2 -24612.987} C_VEL
LIN {X 0,Y 170.852,Z 383.783,A -85,B 0,C 180,E1 -24614.481,E2 -24614.481} C_VEL
LIN {X 0,Y 171.292,Z 378.153,A -85,B 0,C 180,E1 -24615.065,E2 -24615.065} C_VEL
LIN {X 0,Y 172.732,Z 367.701,A -85,B 0,C 180,E1 -24615.663,E2 -24615.663} C_VEL
LIN {X 0,Y 174.955,Z 336.649,A -85,B 0,C 180,E1 -24616.83,E2 -24616.83} C_VEL
LIN {X 0,Y 175.164,Z 330.968,A -85,B 0,C 180,E1 -24617.09,E2 -24617.09} C_VEL
LIN {X 0,Y 174.143,Z 327.406,A -85,B 0,C 180,E1 -24617.663,E2 -24617.663} C_VEL
LIN {X 0,Y 169.286,Z 314.812,A -85,B 0,C 180,E1 -24620.296,E2 -24620.296} C_VEL
LIN {X 0,Y 163.389,Z 302.249,A -85,B 0,C 180,E1 -24623.739,E2 -24623.739} C_VEL
LIN {X 0,Y 158.735,Z 293.8,A -85,B 0,C 180,E1 -24626.752,E2 -24626.752} C_VEL
LIN {X 0,Y 155.989,Z 289.921,A -85,B 0,C 180,E1 -24628.644,E2 -24628.644} C_VEL
LIN {X 0,Y 153.286,Z 286.16,A -85,B 0,C 180,E1 -24630.68,E2 -24630.68} C_VEL
LIN {X 0,Y 150.67,Z 282.711,A -85,B 0,C 180,E1 -24632.836,E2 -24632.836} C_VEL
LIN {X 0,Y 149.849,Z 281.625,A -85,B 0,C 180,E1 -24633.563,E2 -24633.563} C_VEL
LIN {X 0,Y 147.101,Z 278.638,A -85,B 0,C 180,E1 -24636.132,E2 -24636.132} C_VEL
LIN {X 0,Y 146.015,Z 276.65,A -85,B 0,C 180,E1 -24637.351,E2 -24637.351} C_VEL
LIN {X 0,Y 143.513,Z 274.645,A -85,B 0,C 180,E1 -24640.138,E2 -24640.138} C_VEL
LIN {X 0,Y 141.795,Z 271.745,A -85,B 0,C 180,E1 -24642.605,E2 -24642.605} C_VEL
LIN {X 0,Y 141.056,Z 270.92,A -85,B 0,C 180,E1 -24643.723,E2 -24643.723} C_VEL
LIN {X 0,Y 138.473,Z 269.09,A -85,B 0,C 180,E1 -24648.285,E2 -24648.285} C_VEL
LIN {X 0,Y 136.718,Z 265.68,A -85,B 0,C 180,E1 -24654.837,E2 -24654.837} C_VEL
LIN {X 0,Y 137.132,Z 264.972,A -85,B 0,C 180,E1 -24659.998,E2 -24659.998} C_VEL
LIN {X 0,Y 136.709,Z 265.591,A -85,B 0,C 180,E1 -24665.16,E2 -24665.16} C_VEL
LIN {X 0,Y 137.382,Z 267.514,A -85,B 0,C 180,E1 -24669.197,E2 -24669.197} C_VEL
LIN {X 0,Y 139.937,Z 270.328,A -85,B 0,C 180,E1 -24674.914,E2 -24674.914} C_VEL
LIN {X 0,Y 141.747,Z 271.517,A -85,B 0,C 180,E1 -24677.677,E2 -24677.677} C_VEL
LIN {X 0,Y 143.444,Z 274.592,A -85,B 0,C 180,E1 -24680.161,E2 -24680.161} C_VEL
LIN {X 0,Y 146.224,Z 276.98,A -85,B 0,C 180,E1 -24683.265,E2 -24683.265} C_VEL
LIN {X 0,Y 148.483,Z 280.413,A -85,B 0,C 180,E1 -24685.614,E2 -24685.614} C_VEL
LIN {X 0,Y 150.387,Z 282.194,A -85,B 0,C 180,E1 -24687.284,E2 -24687.284} C_VEL
LIN {X 0,Y 152.813,Z 285.711,A -85,B 0,C 180,E1 -24689.345,E2 -24689.345} C_VEL
LIN {X 0,Y 154.096,Z 287.215,A -85,B 0,C 180,E1 -24690.326,E2 -24690.326} C_VEL
LIN {X 0,Y 157.764,Z 292.388,A -85,B 0,C 180,E1 -24692.976,E2 -24692.976} C_VEL
LIN {X 0,Y 161.036,Z 297.109,A -85,B 0,C 180,E1 -24695.103,E2 -24695.103} C_VEL
LIN {X 0,Y 166.416,Z 305.642,A -85,B 0,C 180,E1 -24698.264,E2 -24698.264} C_VEL
LIN {X 0,Y 171.85,Z 315.398,A -85,B 0,C 180,E1 -24701.134,E2 -24701.134} C_VEL
LIN {X 0,Y 176.309,Z 324.483,A -85,B 0,C 180,E1 -24703.31,E2 -24703.31} C_VEL
LIN {X 0,Y 181.534,Z 336.962,A -85,B 0,C 180,E1 -24705.726,E2 -24705.726} C_VEL
LIN {X 0,Y 188.138,Z 352.274,A -85,B 0,C 180,E1 -24708.44,E2 -24708.44} C_VEL
LIN {X 0,Y 195.19,Z 365.92,A -85,B 0,C 180,E1 -24711.133,E2 -24711.133} C_VEL
LIN {X 0,Y 201.415,Z 376.695,A -85,B 0,C 180,E1 -24713.617,E2 -24713.617} C_VEL
LIN {X 0,Y 207.442,Z 385.718,A -85,B 0,C 180,E1 -24715.963,E2 -24715.963} C_VEL
LIN {X 0,Y 215.358,Z 396.067,A -85,B 0,C 180,E1 -24718.939,E2 -24718.939} C_VEL
LIN {X 0,Y 223.899,Z 405.476,A -85,B 0,C 180,E1 -24721.912,E2 -24721.912} C_VEL
LIN {X 0,Y 234.418,Z 414.903,A -85,B 0,C 180,E1 -24725.183,E2 -24725.183} C_VEL
LIN {X 0,Y 246.715,Z 423.801,A -85,B 0,C 180,E1 -24728.551,E2 -24728.551} C_VEL
LIN {X 0,Y 261.029,Z 432.428,A -85,B 0,C 180,E1 -24732.056,E2 -24732.056} C_VEL
LIN {X 0,Y 270.139,Z 437.682,A -85,B 0,C 180,E1 -24734.277,E2 -24734.277} C_VEL
LIN {X 0,Y 278.191,Z 442.264,A -85,B 0,C 180,E1 -24736.294,E2 -24736.294} C_VEL
LIN {X 0,Y 286.626,Z 447.378,A -85,B 0,C 180,E1 -24738.688,E2 -24738.688} C_VEL
LIN {X 0,Y 291.656,Z 450.417,A -85,B 0,C 180,E1 -24740.289,E2 -24740.289} C_VEL
LIN {X 0,Y 295.171,Z 452.887,A -85,B 0,C 180,E1 -24741.787,E2 -24741.787} C_VEL
LIN {X 0,Y 298.238,Z 454.835,A -85,B 0,C 180,E1 -24743.233,E2 -24743.233} C_VEL
LIN {X 0,Y 300.699,Z 456.196,A -85,B 0,C 180,E1 -24744.636,E2 -24744.636} C_VEL
LIN {X 0,Y 302.913,Z 457.248,A -85,B 0,C 180,E1 -24746.067,E2 -24746.067} C_VEL
LIN {X 0,Y 304.424,Z 457.92,A -85,B 0,C 180,E1 -24747.354,E2 -24747.354} C_VEL
LIN {X 0,Y 305.371,Z 458.313,A -85,B 0,C 180,E1 -24748.681,E2 -24748.681} C_VEL
LIN {X 0,Y 305.849,Z 458.398,A -85,B 0,C 180,E1 -24750,E2 -24750} C_VEL
LIN {X 0,Y 305.386,Z 458.313,A -85,B 0,C 180,E1 -24751.319,E2 -24751.319} C_VEL
LIN {X 0,Y 304.446,Z 457.924,A -85,B 0,C 180,E1 -24752.646,E2 -24752.646} C_VEL
LIN {X 0,Y 302.813,Z 457.233,A -85,B 0,C 180,E1 -24753.993,E2 -24753.993} C_VEL
LIN {X 0,Y 300.699,Z 456.226,A -85,B 0,C 180,E1 -24755.364,E2 -24755.364} C_VEL
LIN {X 0,Y 297.467,Z 454.399,A -85,B 0,C 180,E1 -24757.123,E2 -24757.123} C_VEL
LIN {X 0,Y 293.71,Z 451.879,A -85,B 0,C 180,E1 -24758.853,E2 -24758.853} C_VEL
LIN {X 0,Y 291.618,Z 450.419,A -85,B 0,C 180,E1 -24759.712,E2 -24759.712} C_VEL
LIN {X 0,Y 286.624,Z 447.378,A -85,B 0,C 180,E1 -24761.312,E2 -24761.312} C_VEL
LIN {X 0,Y 278.183,Z 442.273,A -85,B 0,C 180,E1 -24763.704,E2 -24763.704} C_VEL
LIN {X 0,Y 270.14,Z 437.678,A -85,B 0,C 180,E1 -24765.724,E2 -24765.724} C_VEL
LIN {X 0,Y 259.187,Z 431.396,A -85,B 0,C 180,E1 -24768.372,E2 -24768.372} C_VEL
LIN {X 0,Y 244.971,Z 422.665,A -85,B 0,C 180,E1 -24771.898,E2 -24771.898} C_VEL
LIN {X 0,Y 233.05,Z 413.782,A -85,B 0,C 180,E1 -24775.22,E2 -24775.22} C_VEL
LIN {X 0,Y 223.392,Z 404.999,A -85,B 0,C 180,E1 -24778.252,E2 -24778.252} C_VEL
LIN {X 0,Y 213.393,Z 393.601,A -85,B 0,C 180,E1 -24781.8,E2 -24781.8} C_VEL
LIN {X 0,Y 205.455,Z 382.805,A -85,B 0,C 180,E1 -24784.82,E2 -24784.82} C_VEL
LIN {X 0,Y 198.974,Z 372.564,A -85,B 0,C 180,E1 -24787.372,E2 -24787.372} C_VEL
LIN {X 0,Y 192.463,Z 360.817,A -85,B 0,C 180,E1 -24789.931,E2 -24789.931} C_VEL
LIN {X 0,Y 186.275,Z 348.363,A -85,B 0,C 180,E1 -24792.274,E2 -24792.274} C_VEL
LIN {X 0,Y 177.745,Z 327.775,A -85,B 0,C 180,E1 -24796.009,E2 -24796.009} C_VEL
LIN {X 0,Y 172.771,Z 317.082,A -85,B 0,C 180,E1 -24798.411,E2 -24798.411} C_VEL
LIN {X 0,Y 167.554,Z 307.615,A -85,B 0,C 180,E1 -24801.109,E2 -24801.109} C_VEL
LIN {X 0,Y 161.865,Z 298.285,A -85,B 0,C 180,E1 -24804.39,E2 -24804.39} C_VEL
LIN {X 0,Y 156.578,Z 290.646,A -85,B 0,C 180,E1 -24807.852,E2 -24807.852} C_VEL
LIN {X 0,Y 153.303,Z 286.159,A -85,B 0,C 180,E1 -24810.287,E2 -24810.287} C_VEL
LIN {X 0,Y 150.724,Z 282.854,A -85,B 0,C 180,E1 -24812.4,E2 -24812.4} C_VEL
LIN {X 0,Y 149.975,Z 281.723,A -85,B 0,C 180,E1 -24813.075,E2 -24813.075} C_VEL
LIN {X 0,Y 147.365,Z 279.011,A -85,B 0,C 180,E1 -24815.478,E2 -24815.478} C_VEL
LIN {X 0,Y 146.008,Z 276.622,A -85,B 0,C 180,E1 -24816.979,E2 -24816.979} C_VEL
LIN {X 0,Y 143.518,Z 274.685,A -85,B 0,C 180,E1 -24819.744,E2 -24819.744} C_VEL
LIN {X 0,Y 141.9,Z 271.91,A -85,B 0,C 180,E1 -24822.063,E2 -24822.063} C_VEL
LIN {X 0,Y 141.283,Z 271.051,A -85,B 0,C 180,E1 -24823.009,E2 -24823.009} C_VEL
LIN {X 0,Y 138.201,Z 268.763,A -85,B 0,C 180,E1 -24828.536,E2 -24828.536} C_VEL
LIN {X 0,Y 136.718,Z 265.819,A -85,B 0,C 180,E1 -24834.101,E2 -24834.101} C_VEL
LIN {X 0,Y 137.029,Z 265.025,A -85,B 0,C 180,E1 -24839.267,E2 -24839.267} C_VEL
LIN {X 0,Y 136.849,Z 265.136,A -85,B 0,C 180,E1 -24842.209,E2 -24842.209} C_VEL
LIN {X 0,Y 136.802,Z 266.131,A -85,B 0,C 180,E1 -24846.269,E2 -24846.269} C_VEL
LIN {X 0,Y 139.735,Z 270.238,A -85,B 0,C 180,E1 -24854.195,E2 -24854.195} C_VEL
LIN {X 0,Y 141.694,Z 271.485,A -85,B 0,C 180,E1 -24857.222,E2 -24857.222} C_VEL
LIN {X 0,Y 143.382,Z 274.477,A -85,B 0,C 180,E1 -24859.695,E2 -24859.695} C_VEL
LIN {X 0,Y 145.756,Z 276.496,A -85,B 0,C 180,E1 -24862.387,E2 -24862.387} C_VEL
LIN {X 0,Y 146.511,Z 277.596,A -85,B 0,C 180,E1 -24863.22,E2 -24863.22} C_VEL
LIN {X 0,Y 148.805,Z 280.717,A -85,B 0,C 180,E1 -24865.525,E2 -24865.525} C_VEL
LIN {X 0,Y 150.415,Z 282.296,A -85,B 0,C 180,E1 -24866.933,E2 -24866.933} C_VEL
LIN {X 0,Y 153.069,Z 285.914,A -85,B 0,C 180,E1 -24869.154,E2 -24869.154} C_VEL
LIN {X 0,Y 157.462,Z 291.937,A -85,B 0,C 180,E1 -24872.386,E2 -24872.386} C_VEL
LIN {X 0,Y 159.864,Z 295.817,A -85,B 0,C 180,E1 -24874.014,E2 -24874.014} C_VEL
LIN {X 0,Y 164.045,Z 303.574,A -85,B 0,C 180,E1 -24876.665,E2 -24876.665} C_VEL
LIN {X 0,Y 170.106,Z 316.712,A -85,B 0,C 180,E1 -24880.155,E2 -24880.155} C_VEL
LIN {X 0,Y 174.976,Z 329.733,A -85,B 0,C 180,E1 -24882.771,E2 -24882.771} C_VEL
LIN {X 0,Y 175.208,Z 333.073,A -85,B 0,C 180,E1 -24883.049,E2 -24883.049} C_VEL
LIN {X 0,Y 172.685,Z 367.897,A -85,B 0,C 180,E1 -24884.33,E2 -24884.33} C_VEL
LIN {X 0,Y 170.956,Z 380.367,A -85,B 0,C 180,E1 -24885.086,E2 -24885.086} C_VEL
LIN {X 0,Y 167.941,Z 393.954,A -85,B 0,C 180,E1 -24886.331,E2 -24886.331} C_VEL
LIN {X 0,Y 165.242,Z 403.464,A -85,B 0,C 180,E1 -24887.532,E2 -24887.532} C_VEL
LIN {X 0,Y 162.124,Z 412.735,A -85,B 0,C 180,E1 -24889.031,E2 -24889.031} C_VEL
LIN {X 0,Y 158.687,Z 421.676,A -85,B 0,C 180,E1 -24890.868,E2 -24890.868} C_VEL
LIN {X 0,Y 154.954,Z 430.199,A -85,B 0,C 180,E1 -24893.062,E2 -24893.062} C_VEL
LIN {X 0,Y 151.441,Z 437.412,A -85,B 0,C 180,E1 -24895.355,E2 -24895.355} C_VEL
LIN {X 0,Y 148.283,Z 443.612,A -85,B 0,C 180,E1 -24897.778,E2 -24897.778} C_VEL
LIN {X 0,Y 144.831,Z 450.151,A -85,B 0,C 180,E1 -24900.971,E2 -24900.971} C_VEL
LIN {X 0,Y 142.346,Z 454.654,A -85,B 0,C 180,E1 -24903.618,E2 -24903.618} C_VEL
LIN {X 0,Y 139.066,Z 460.144,A -85,B 0,C 180,E1 -24907.727,E2 -24907.727} C_VEL
LIN {X 0,Y 136.493,Z 464.47,A -85,B 0,C 180,E1 -24912.005,E2 -24912.005} C_VEL
LIN {X 0,Y 135.326,Z 466.844,A -85,B 0,C 180,E1 -24914.95,E2 -24914.95} C_VEL
LIN {X 0,Y 134.433,Z 468.648,A -85,B 0,C 180,E1 -24917.93,E2 -24917.93} C_VEL
LIN {X 0,Y 133.542,Z 471.109,A -85,B 0,C 180,E1 -24923.958,E2 -24923.958} C_VEL
LIN {X 0,Y 133.414,Z 471.704,A -85,B 0,C 180,E1 -24926.98,E2 -24926.98} C_VEL
LIN {X 0,Y 133.536,Z 471.864,A -85,B 0,C 180,E1 -24930,E2 -24930} C_VEL
LIN {X 0,Y 133.4,Z 471.703,A -85,B 0,C 180,E1 -24933.02,E2 -24933.02} C_VEL
LIN {X 0,Y 133.462,Z 471.107,A -85,B 0,C 180,E1 -24936.045,E2 -24936.045} C_VEL
LIN {X 0,Y 134.381,Z 468.647,A -85,B 0,C 180,E1 -24942.075,E2 -24942.075} C_VEL
LIN {X 0,Y 135.867,Z 465.69,A -85,B 0,C 180,E1 -24946.529,E2 -24946.529} C_VEL
LIN {X 0,Y 138.119,Z 461.698,A -85,B 0,C 180,E1 -24950.866,E2 -24950.866} C_VEL
LIN {X 0,Y 141.119,Z 456.567,A -85,B 0,C 180,E1 -24955.044,E2 -24955.044} C_VEL
LIN {X 0,Y 144.184,Z 451.318,A -85,B 0,C 180,E1 -24958.368,E2 -24958.368} C_VEL
LIN {X 0,Y 147.531,Z 444.988,A -85,B 0,C 180,E1 -24961.602,E2 -24961.602} C_VEL
LIN {X 0,Y 150.627,Z 439.039,A -85,B 0,C 180,E1 -24964.049,E2 -24964.049} C_VEL
LIN {X 0,Y 154.055,Z 432.117,A -85,B 0,C 180,E1 -24966.374,E2 -24966.374} C_VEL
LIN {X 0,Y 157.706,Z 423.943,A -85,B 0,C 180,E1 -24968.601,E2 -24968.601} C_VEL
LIN {X 0,Y 161.083,Z 415.435,A -85,B 0,C 180,E1 -24970.465,E2 -24970.465} C_VEL
LIN {X 0,Y 164.176,Z 406.66,A -85,B 0,C 180,E1 -24971.996,E2 -24971.996} C_VEL
LIN {X 0,Y 167.139,Z 396.974,A -85,B 0,C 180,E1 -24973.308,E2 -24973.308} C_VEL
LIN {X 0,Y 169.31,Z 388.183,A -85,B 0,C 180,E1 -24974.257,E2 -24974.257} C_VEL
LIN {X 0,Y 171.292,Z 378.153,A -85,B 0,C 180,E1 -24975.065,E2 -24975.065} C_VEL
LIN {X 0,Y 171.742,Z 371.514,A -85,B 0,C 180,E1 -24975.69,E2 -24975.69} C_VEL
LIN {X 0,Y 169.435,Z 353.848,A -85,B 0,C 180,E1 -24977.785,E2 -24977.785} C_VEL
LIN {X 0,Y 169.369,Z 348.036,A -85,B 0,C 180,E1 -24978.158,E2 -24978.158} C_VEL
LIN {X 0,Y 170.338,Z 332.721,A -85,B 0,C 180,E1 -24978.745,E2 -24978.745} C_VEL
LIN {X 0,Y 165.582,Z 319.709,A -85,B 0,C 180,E1 -24981.521,E2 -24981.521} C_VEL
LIN {X 0,Y 159.833,Z 307.015,A -85,B 0,C 180,E1 -24985.135,E2 -24985.135} C_VEL
LIN {X 0,Y 155.651,Z 299.186,A -85,B 0,C 180,E1 -24988.052,E2 -24988.052} C_VEL
LIN {X 0,Y 153.114,Z 295.508,A -85,B 0,C 180,E1 -24989.93,E2 -24989.93} C_VEL
LIN {X 0,Y 150.812,Z 292.211,A -85,B 0,C 180,E1 -24991.786,E2 -24991.786} C_VEL
LIN {X 0,Y 147.804,Z 288.052,A -85,B 0,C 180,E1 -24994.476,E2 -24994.476} C_VEL
LIN {X 0,Y 144.966,Z 284.679,A -85,B 0,C 180,E1 -24997.331,E2 -24997.331} C_VEL
LIN {X 0,Y 143.985,Z 283.15,A -85,B 0,C 180,E1 -24998.476,E2 -24998.476} C_VEL
LIN {X 0,Y 141.351,Z 280.483,A -85,B 0,C 180,E1 -25001.753,E2 -25001.753} C_VEL
LIN {X 0,Y 139.984,Z 277.918,A -85,B 0,C 180,E1 -25003.969,E2 -25003.969} C_VEL
LIN {X 0,Y 137.256,Z 275.846,A -85,B 0,C 180,E1 -25009.04,E2 -25009.04} C_VEL
LIN {X 0,Y 135.517,Z 272.546,A -85,B 0,C 180,E1 -25015.537,E2 -25015.537} C_VEL
LIN {X 0,Y 135.162,Z 271.802,A -85,B 0,C 180,E1 -25019.998,E2 -25019.998} C_VEL
LIN {X 0,Y 135.574,Z 272.667,A -85,B 0,C 180,E1 -25025.203,E2 -25025.203} C_VEL
LIN {X 0,Y 138.585,Z 277.13,A -85,B 0,C 180,E1 -25034.124,E2 -25034.124} C_VEL
LIN {X 0,Y 140.223,Z 278.198,A -85,B 0,C 180,E1 -25036.795,E2 -25036.795} C_VEL
LIN {X 0,Y 141.987,Z 281.371,A -85,B 0,C 180,E1 -25039.517,E2 -25039.517} C_VEL
LIN {X 0,Y 144.525,Z 283.788,A -85,B 0,C 180,E1 -25042.519,E2 -25042.519} C_VEL
LIN {X 0,Y 146.782,Z 287.095,A -85,B 0,C 180,E1 -25044.956,E2 -25044.956} C_VEL
LIN {X 0,Y 148.375,Z 288.847,A -85,B 0,C 180,E1 -25046.445,E2 -25046.445} C_VEL
LIN {X 0,Y 151.123,Z 292.551,A -85,B 0,C 180,E1 -25048.846,E2 -25048.846} C_VEL
LIN {X 0,Y 155.471,Z 298.878,A -85,B 0,C 180,E1 -25052.198,E2 -25052.198} C_VEL
LIN {X 0,Y 159.21,Z 304.478,A -85,B 0,C 180,E1 -25054.729,E2 -25054.729} C_VEL
LIN {X 0,Y 165.407,Z 315.133,A -85,B 0,C 180,E1 -25058.472,E2 -25058.472} C_VEL
LIN {X 0,Y 171.096,Z 326.446,A -85,B 0,C 180,E1 -25061.535,E2 -25061.535} C_VEL
LIN {X 0,Y 176.441,Z 339.286,A -85,B 0,C 180,E1 -25064.212,E2 -25064.212} C_VEL
LIN {X 0,Y 182.744,Z 354.769,A -85,B 0,C 180,E1 -25067.044,E2 -25067.044} C_VEL
LIN {X 0,Y 188.869,Z 367.542,A -85,B 0,C 180,E1 -25069.712,E2 -25069.712} C_VEL
LIN {X 0,Y 193.871,Z 376.937,A -85,B 0,C 180,E1 -25071.956,E2 -25071.956} C_VEL
LIN {X 0,Y 200.114,Z 387.265,A -85,B 0,C 180,E1 -25074.738,E2 -25074.738} C_VEL
LIN {X 0,Y 206.117,Z 395.723,A -85,B 0,C 180,E1 -25077.266,E2 -25077.266} C_VEL
LIN {X 0,Y 213.176,Z 404.346,A -85,B 0,C 180,E1 -25080.067,E2 -25080.067} C_VEL
LIN {X 0,Y 221.007,Z 412.463,A -85,B 0,C 180,E1 -25082.92,E2 -25082.92} C_VEL
LIN {X 0,Y 230.712,Z 420.572,A -85,B 0,C 180,E1 -25086.043,E2 -25086.043} C_VEL
LIN {X 0,Y 240.949,Z 427.621,A -85,B 0,C 180,E1 -25088.964,E2 -25088.964} C_VEL
LIN {X 0,Y 253.864,Z 435.09,A -85,B 0,C 180,E1 -25092.27,E2 -25092.27} C_VEL
LIN {X 0,Y 262.831,Z 439.891,A -85,B 0,C 180,E1 -25094.491,E2 -25094.491} C_VEL
LIN {X 0,Y 270.741,Z 444.062,A -85,B 0,C 180,E1 -25096.489,E2 -25096.489} C_VEL
LIN {X 0,Y 279.293,Z 448.808,A -85,B 0,C 180,E1 -25098.92,E2 -25098.92} C_VEL
LIN {X 0,Y 284.878,Z 451.891,A -85,B 0,C 180,E1 -25100.678,E2 -25100.678} C_VEL
LIN {X 0,Y 288.785,Z 454.426,A -85,B 0,C 180,E1 -25102.309,E2 -25102.309} C_VEL
LIN {X 0,Y 293.096,Z 457.053,A -85,B 0,C 180,E1 -25104.496,E2 -25104.496} C_VEL
LIN {X 0,Y 295.828,Z 458.446,A -85,B 0,C 180,E1 -25106.18,E2 -25106.18} C_VEL
LIN {X 0,Y 297.186,Z 459.071,A -85,B 0,C 180,E1 -25107.289,E2 -25107.289} C_VEL
LIN {X 0,Y 298.295,Z 459.489,A -85,B 0,C 180,E1 -25108.65,E2 -25108.65} C_VEL
LIN {X 0,Y 298.858,Z 459.591,A -85,B 0,C 180,E1 -25110,E2 -25110} C_VEL
LIN {X 0,Y 298.31,Z 459.493,A -85,B 0,C 180,E1 -25111.35,E2 -25111.35} C_VEL
LIN {X 0,Y 297.203,Z 459.083,A -85,B 0,C 180,E1 -25112.711,E2 -25112.711} C_VEL
LIN {X 0,Y 295.39,Z 458.282,A -85,B 0,C 180,E1 -25114.093,E2 -25114.093} C_VEL
LIN {X 0,Y 293.097,Z 457.06,A -85,B 0,C 180,E1 -25115.504,E2 -25115.504} C_VEL
LIN {X 0,Y 290.289,Z 455.44,A -85,B 0,C 180,E1 -25116.97,E2 -25116.97} C_VEL
LIN {X 0,Y 287.045,Z 453.311,A -85,B 0,C 180,E1 -25118.448,E2 -25118.448} C_VEL
LIN {X 0,Y 284.873,Z 451.901,A -85,B 0,C 180,E1 -25119.317,E2 -25119.317} C_VEL
LIN {X 0,Y 277.143,Z 447.642,A -85,B 0,C 180,E1 -25121.705,E2 -25121.705} C_VEL
LIN {X 0,Y 270.724,Z 444.063,A -85,B 0,C 180,E1 -25123.511,E2 -25123.511} C_VEL
LIN {X 0,Y 259.098,Z 437.891,A -85,B 0,C 180,E1 -25126.445,E2 -25126.445} C_VEL
LIN {X 0,Y 246.271,Z 430.777,A -85,B 0,C 180,E1 -25129.656,E2 -25129.656} C_VEL
LIN {X 0,Y 234.066,Z 422.975,A -85,B 0,C 180,E1 -25132.975,E2 -25132.975} C_VEL
LIN {X 0,Y 224.1,Z 415.202,A -85,B 0,C 180,E1 -25136.043,E2 -25136.043} C_VEL
LIN {X 0,Y 216.378,Z 407.873,A -85,B 0,C 180,E1 -25138.724,E2 -25138.724} C_VEL
LIN {X 0,Y 208.595,Z 398.932,A -85,B 0,C 180,E1 -25141.718,E2 -25141.718} C_VEL
LIN {X 0,Y 202.21,Z 390.338,A -85,B 0,C 180,E1 -25144.368,E2 -25144.368} C_VEL
LIN {X 0,Y 195.984,Z 380.734,A -85,B 0,C 180,E1 -25147.073,E2 -25147.073} C_VEL
LIN {X 0,Y 190.142,Z 370.019,A -85,B 0,C 180,E1 -25149.714,E2 -25149.714} C_VEL
LIN {X 0,Y 184.736,Z 359.047,A -85,B 0,C 180,E1 -25152.113,E2 -25152.113} C_VEL
LIN {X 0,Y 177.875,Z 343.157,A -85,B 0,C 180,E1 -25155.094,E2 -25155.094} C_VEL
LIN {X 0,Y 173.004,Z 330.836,A -85,B 0,C 180,E1 -25157.486,E2 -25157.486} C_VEL
LIN {X 0,Y 168.522,Z 321.129,A -85,B 0,C 180,E1 -25159.814,E2 -25159.814} C_VEL
LIN {X 0,Y 163.445,Z 311.671,A -85,B 0,C 180,E1 -25162.654,E2 -25162.654} C_VEL
LIN {X 0,Y 158.563,Z 303.53,A -85,B 0,C 180,E1 -25165.687,E2 -25165.687} C_VEL
LIN {X 0,Y 154.053,Z 296.711,A -85,B 0,C 180,E1 -25168.848,E2 -25168.848} C_VEL
LIN {X 0,Y 150.746,Z 292.161,A -85,B 0,C 180,E1 -25171.455,E2 -25171.455} C_VEL
LIN {X 0,Y 147.65,Z 287.939,A -85,B 0,C 180,E1 -25174.231,E2 -25174.231} C_VEL
LIN {X 0,Y 145.008,Z 284.713,A -85,B 0,C 180,E1 -25176.906,E2 -25176.906} C_VEL
LIN {X 0,Y 144.025,Z 283.176,A -85,B 0,C 180,E1 -25178.052,E2 -25178.052} C_VEL
LIN {X 0,Y 141.616,Z 280.86,A -85,B 0,C 180,E1 -25180.995,E2 -25180.995} C_VEL
LIN {X 0,Y 139.978,Z 277.902,A -85,B 0,C 180,E1 -25183.597,E2 -25183.597} C_VEL
LIN {X 0,Y 137.107,Z 275.687,A -85,B 0,C 180,E1 -25189.022,E2 -25189.022} C_VEL
LIN {X 0,Y 135.512,Z 272.567,A -85,B 0,C 180,E1 -25195.167,E2 -25195.167} C_VEL
LIN {X 0,Y 135.162,Z 271.799,A -85,B 0,C 180,E1 -25200.002,E2 -25200.002} C_VEL
LIN {X 0,Y 135.638,Z 272.81,A -85,B 0,C 180,E1 -25205.204,E2 -25205.204} C_VEL
LIN {X 0,Y 138.685,Z 277.231,A -85,B 0,C 180,E1 -25213.93,E2 -25213.93} C_VEL
LIN {X 0,Y 140.196,Z 278.216,A -85,B 0,C 180,E1 -25216.38,E2 -25216.38} C_VEL
LIN {X 0,Y 141.997,Z 281.347,A -85,B 0,C 180,E1 -25219.143,E2 -25219.143} C_VEL
LIN {X 0,Y 144.457,Z 283.737,A -85,B 0,C 180,E1 -25222.064,E2 -25222.064} C_VEL
LIN {X 0,Y 146.772,Z 287.089,A -85,B 0,C 180,E1 -25224.565,E2 -25224.565} C_VEL
LIN {X 0,Y 148.403,Z 288.869,A -85,B 0,C 180,E1 -25226.088,E2 -25226.088} C_VEL
LIN {X 0,Y 151.186,Z 292.572,A -85,B 0,C 180,E1 -25228.51,E2 -25228.51} C_VEL
LIN {X 0,Y 156.061,Z 299.759,A -85,B 0,C 180,E1 -25232.235,E2 -25232.235} C_VEL
LIN {X 0,Y 160.675,Z 308.748,A -85,B 0,C 180,E1 -25235.421,E2 -25235.421} C_VEL
LIN {X 0,Y 166.362,Z 321.627,A -85,B 0,C 180,E1 -25238.942,E2 -25238.942} C_VEL
LIN {X 0,Y 170.317,Z 332.639,A -85,B 0,C 180,E1 -25241.242,E2 -25241.242} C_VEL
LIN {X 0,Y 169.645,Z 343.638,A -85,B 0,C 180,E1 -25241.672,E2 -25241.672} C_VEL
LIN {X 0,Y 167.706,Z 368.624,A -85,B 0,C 180,E1 -25242.64,E2 -25242.64} C_VEL
LIN {X 0,Y 165.683,Z 381.925,A -85,B 0,C 180,E1 -25243.481,E2 -25243.481} C_VEL
LIN {X 0,Y 162.889,Z 393.761,A -85,B 0,C 180,E1 -25244.61,E2 -25244.61} C_VEL
LIN {X 0,Y 160.085,Z 403.272,A -85,B 0,C 180,E1 -25245.818,E2 -25245.818} C_VEL
LIN {X 0,Y 156.835,Z 412.542,A -85,B 0,C 180,E1 -25247.33,E2 -25247.33} C_VEL
LIN {X 0,Y 153.23,Z 421.483,A -85,B 0,C 180,E1 -25249.188,E2 -25249.188} C_VEL
LIN {X 0,Y 149.325,Z 430.006,A -85,B 0,C 180,E1 -25251.42,E2 -25251.42} C_VEL
LIN {X 0,Y 145.65,Z 437.219,A -85,B 0,C 180,E1 -25253.765,E2 -25253.765} C_VEL
LIN {X 0,Y 142.318,Z 443.419,A -85,B 0,C 180,E1 -25256.252,E2 -25256.252} C_VEL
LIN {X 0,Y 138.634,Z 449.958,A -85,B 0,C 180,E1 -25259.539,E2 -25259.539} C_VEL
LIN {X 0,Y 136.018,Z 454.461,A -85,B 0,C 180,E1 -25262.288,E2 -25262.288} C_VEL
LIN {X 0,Y 132.497,Z 459.951,A -85,B 0,C 180,E1 -25266.558,E2 -25266.558} C_VEL
LIN {X 0,Y 129.723,Z 464.276,A -85,B 0,C 180,E1 -25271.031,E2 -25271.031} C_VEL
LIN {X 0,Y 128.444,Z 466.65,A -85,B 0,C 180,E1 -25274.123,E2 -25274.123} C_VEL
LIN {X 0,Y 127.464,Z 468.455,A -85,B 0,C 180,E1 -25277.259,E2 -25277.259} C_VEL
LIN {X 0,Y 126.463,Z 470.916,A -85,B 0,C 180,E1 -25283.619,E2 -25283.619} C_VEL
LIN {X 0,Y 126.317,Z 471.511,A -85,B 0,C 180,E1 -25286.811,E2 -25286.811} C_VEL
LIN {X 0,Y 126.431,Z 471.671,A -85,B 0,C 180,E1 -25290,E2 -25290} C_VEL
LIN {X 0,Y 126.305,Z 471.51,A -85,B 0,C 180,E1 -25293.19,E2 -25293.19} C_VEL
LIN {X 0,Y 126.405,Z 470.914,A -85,B 0,C 180,E1 -25296.384,E2 -25296.384} C_VEL
LIN {X 0,Y 127.422,Z 468.453,A -85,B 0,C 180,E1 -25302.745,E2 -25302.745} C_VEL
LIN {X 0,Y 129.046,Z 465.496,A -85,B 0,C 180,E1 -25307.43,E2 -25307.43} C_VEL
LIN {X 0,Y 131.484,Z 461.505,A -85,B 0,C 180,E1 -25311.972,E2 -25311.972} C_VEL
LIN {X 0,Y 134.707,Z 456.374,A -85,B 0,C 180,E1 -25316.325,E2 -25316.325} C_VEL
LIN {X 0,Y 138.634,Z 449.958,A -85,B 0,C 180,E1 -25320.461,E2 -25320.461} C_VEL
LIN {X 0,Y 143.116,Z 442.035,A -85,B 0,C 180,E1 -25324.383,E2 -25324.383} C_VEL
LIN {X 0,Y 147.45,Z 433.841,A -85,B 0,C 180,E1 -25327.424,E2 -25327.424} C_VEL
LIN {X 0,Y 151.728,Z 424.884,A -85,B 0,C 180,E1 -25329.992,E2 -25329.992} C_VEL
LIN {X 0,Y 155.228,Z 416.593,A -85,B 0,C 180,E1 -25331.898,E2 -25331.898} C_VEL
LIN {X 0,Y 158.952,Z 406.532,A -85,B 0,C 180,E1 -25333.697,E2 -25333.697} C_VEL
LIN {X 0,Y 162.038,Z 396.781,A -85,B 0,C 180,E1 -25335.033,E2 -25335.033} C_VEL
LIN {X 0,Y 164.305,Z 387.99,A -85,B 0,C 180,E1 -25335.983,E2 -25335.983} C_VEL
LIN {X 0,Y 166.392,Z 377.667,A -85,B 0,C 180,E1 -25336.819,E2 -25336.819} C_VEL
LIN {X 0,Y 167.865,Z 367.307,A -85,B 0,C 180,E1 -25337.407,E2 -25337.407} C_VEL
LIN {X 0,Y 169.369,Z 348.036,A -85,B 0,C 180,E1 -25338.158,E2 -25338.158} C_VEL
LIN {X 0,Y 169.184,Z 344.223,A -85,B 0,C 180,E1 -25338.465,E2 -25338.465} C_VEL
LIN {X 0,Y 168.332,Z 340.697,A -85,B 0,C 180,E1 -25339.015,E2 -25339.015} C_VEL
LIN {X 0,Y 163.866,Z 329.997,A -85,B 0,C 180,E1 -25341.564,E2 -25341.564} C_VEL
LIN {X 0,Y 160.687,Z 321.634,A -85,B 0,C 180,E1 -25343.615,E2 -25343.615} C_VEL
LIN {X 0,Y 156.277,Z 311.559,A -85,B 0,C 180,E1 -25346.666,E2 -25346.666} C_VEL
LIN {X 0,Y 152.673,Z 304.621,A -85,B 0,C 180,E1 -25349.385,E2 -25349.385} C_VEL
LIN {X 0,Y 148.625,Z 298.495,A -85,B 0,C 180,E1 -25352.734,E2 -25352.734} C_VEL
LIN {X 0,Y 145.581,Z 294.28,A -85,B 0,C 180,E1 -25355.623,E2 -25355.623} C_VEL
LIN {X 0,Y 142.867,Z 290.66,A -85,B 0,C 180,E1 -25358.603,E2 -25358.603} C_VEL
LIN {X 0,Y 142.094,Z 289.647,A -85,B 0,C 180,E1 -25359.547,E2 -25359.547} C_VEL
LIN {X 0,Y 139.433,Z 286.434,A -85,B 0,C 180,E1 -25363.226,E2 -25363.226} C_VEL
LIN {X 0,Y 138.578,Z 284.735,A -85,B 0,C 180,E1 -25364.745,E2 -25364.745} C_VEL
LIN {X 0,Y 135.958,Z 282.493,A -85,B 0,C 180,E1 -25370.084,E2 -25370.084} C_VEL
LIN {X 0,Y 134.54,Z 279.448,A -85,B 0,C 180,E1 -25376.254,E2 -25376.254} C_VEL
LIN {X 0,Y 134.296,Z 278.854,A -85,B 0,C 180,E1 -25379.998,E2 -25379.998} C_VEL
LIN {X 0,Y 134.684,Z 279.781,A -85,B 0,C 180,E1 -25385.144,E2 -25385.144} C_VEL
LIN {X 0,Y 137.333,Z 283.991,A -85,B 0,C 180,E1 -25393.463,E2 -25393.463} C_VEL
LIN {X 0,Y 138.781,Z 284.981,A -85,B 0,C 180,E1 -25395.982,E2 -25395.982} C_VEL
LIN {X 0,Y 140.743,Z 288.383,A -85,B 0,C 180,E1 -25399.127,E2 -25399.127} C_VEL
LIN {X 0,Y 142.781,Z 290.445,A -85,B 0,C 180,E1 -25401.662,E2 -25401.662} C_VEL
LIN {X 0,Y 145.126,Z 293.792,A -85,B 0,C 180,E1 -25404.305,E2 -25404.305} C_VEL
LIN {X 0,Y 146.417,Z 295.415,A -85,B 0,C 180,E1 -25405.593,E2 -25405.593} C_VEL
LIN {X 0,Y 149.861,Z 300.373,A -85,B 0,C 180,E1 -25408.729,E2 -25408.729} C_VEL
LIN {X 0,Y 154.295,Z 306.941,A -85,B 0,C 180,E1 -25412.193,E2 -25412.193} C_VEL
LIN {X 0,Y 159.348,Z 315.525,A -85,B 0,C 180,E1 -25415.651,E2 -25415.651} C_VEL
LIN {X 0,Y 164.128,Z 324.642,A -85,B 0,C 180,E1 -25418.564,E2 -25418.564} C_VEL
LIN {X 0,Y 168.201,Z 333.484,A -85,B 0,C 180,E1 -25420.855,E2 -25420.855} C_VEL
LIN {X 0,Y 172.686,Z 345.064,A -85,B 0,C 180,E1 -25423.254,E2 -25423.254} C_VEL
LIN {X 0,Y 178.66,Z 360.02,A -85,B 0,C 180,E1 -25426.184,E2 -25426.184} C_VEL
LIN {X 0,Y 182.692,Z 369.037,A -85,B 0,C 180,E1 -25428.186,E2 -25428.186} C_VEL
LIN {X 0,Y 187.19,Z 378.262,A -85,B 0,C 180,E1 -25430.489,E2 -25430.489} C_VEL
LIN {X 0,Y 191.702,Z 386.641,A -85,B 0,C 180,E1 -25432.792,E2 -25432.792} C_VEL
LIN {X 0,Y 197.734,Z 396.163,A -85,B 0,C 180,E1 -25435.725,E2 -25435.725} C_VEL
LIN {X 0,Y 205.269,Z 406.035,A -85,B 0,C 180,E1 -25439.098,E2 -25439.098} C_VEL
LIN {X 0,Y 211.901,Z 413.356,A -85,B 0,C 180,E1 -25441.803,E2 -25441.803} C_VEL
LIN {X 0,Y 221.662,Z 422.022,A -85,B 0,C 180,E1 -25445.313,E2 -25445.313} C_VEL
LIN {X 0,Y 233.449,Z 430.237,A -85,B 0,C 180,E1 -25448.945,E2 -25448.945} C_VEL
LIN {X 0,Y 246.815,Z 437.708,A -85,B 0,C 180,E1 -25452.532,E2 -25452.532} C_VEL
LIN {X 0,Y 255.099,Z 441.849,A -85,B 0,C 180,E1 -25454.63,E2 -25454.63} C_VEL
LIN {X 0,Y 263.493,Z 445.924,A -85,B 0,C 180,E1 -25456.787,E2 -25456.787} C_VEL
LIN {X 0,Y 271.914,Z 450.157,A -85,B 0,C 180,E1 -25459.157,E2 -25459.157} C_VEL
LIN {X 0,Y 278.669,Z 453.543,A -85,B 0,C 180,E1 -25461.297,E2 -25461.297} C_VEL
LIN {X 0,Y 283.095,Z 456.134,A -85,B 0,C 180,E1 -25463.221,E2 -25463.221} C_VEL
LIN {X 0,Y 285.269,Z 457.404,A -85,B 0,C 180,E1 -25464.345,E2 -25464.345} C_VEL
LIN {X 0,Y 288.728,Z 459.152,A -85,B 0,C 180,E1 -25466.354,E2 -25466.354} C_VEL
LIN {X 0,Y 289.848,Z 459.633,A -85,B 0,C 180,E1 -25467.22,E2 -25467.22} C_VEL
LIN {X 0,Y 291.105,Z 460.139,A -85,B 0,C 180,E1 -25468.617,E2 -25468.617} C_VEL
LIN {X 0,Y 291.776,Z 460.284,A -85,B 0,C 180,E1 -25470,E2 -25470} C_VEL
LIN {X 0,Y 291.12,Z 460.142,A -85,B 0,C 180,E1 -25471.383,E2 -25471.383} C_VEL
LIN {X 0,Y 289.859,Z 459.633,A -85,B 0,C 180,E1 -25472.779,E2 -25472.779} C_VEL
LIN {X 0,Y 287.806,Z 458.719,A -85,B 0,C 180,E1 -25474.201,E2 -25474.201} C_VEL
LIN {X 0,Y 285.267,Z 457.404,A -85,B 0,C 180,E1 -25475.655,E2 -25475.655} C_VEL
LIN {X 0,Y 282.289,Z 455.692,A -85,B 0,C 180,E1 -25477.151,E2 -25477.151} C_VEL
LIN {X 0,Y 278.655,Z 453.543,A -85,B 0,C 180,E1 -25478.704,E2 -25478.704} C_VEL
LIN {X 0,Y 271.905,Z 450.177,A -85,B 0,C 180,E1 -25480.833,E2 -25480.833} C_VEL
LIN {X 0,Y 263.492,Z 445.928,A -85,B 0,C 180,E1 -25483.212,E2 -25483.212} C_VEL
LIN {X 0,Y 251.752,Z 440.201,A -85,B 0,C 180,E1 -25486.21,E2 -25486.21} C_VEL
LIN {X 0,Y 238.725,Z 433.329,A -85,B 0,C 180,E1 -25489.601,E2 -25489.601} C_VEL
LIN {X 0,Y 225.821,Z 425.138,A -85,B 0,C 180,E1 -25493.353,E2 -25493.353} C_VEL
LIN {X 0,Y 216.155,Z 417.408,A -85,B 0,C 180,E1 -25496.608,E2 -25496.608} C_VEL
LIN {X 0,Y 207.163,Z 408.238,A -85,B 0,C 180,E1 -25500.112,E2 -25500.112} C_VEL
LIN {X 0,Y 199.766,Z 399.033,A -85,B 0,C 180,E1 -25503.329,E2 -25503.329} C_VEL
LIN {X 0,Y 193.737,Z 390.086,A -85,B 0,C 180,E1 -25506.184,E2 -25506.184} C_VEL
LIN {X 0,Y 188.906,Z 381.63,A -85,B 0,C 180,E1 -25508.624,E2 -25508.624} C_VEL
LIN {X 0,Y 183.654,Z 371.106,A -85,B 0,C 180,E1 -25511.325,E2 -25511.325} C_VEL
LIN {X 0,Y 178.822,Z 360.367,A -85,B 0,C 180,E1 -25513.768,E2 -25513.768} C_VEL
LIN {X 0,Y 172.369,Z 344.246,A -85,B 0,C 180,E1 -25516.908,E2 -25516.908} C_VEL
LIN {X 0,Y 168.113,Z 333.27,A -85,B 0,C 180,E1 -25519.193,E2 -25519.193} C_VEL
LIN {X 0,Y 164.061,Z 324.482,A -85,B 0,C 180,E1 -25521.476,E2 -25521.476} C_VEL
LIN {X 0,Y 159.143,Z 315.204,A -85,B 0,C 180,E1 -25524.478,E2 -25524.478} C_VEL
LIN {X 0,Y 154.104,Z 306.619,A -85,B 0,C 180,E1 -25527.949,E2 -25527.949} C_VEL
LIN {X 0,Y 148.794,Z 298.713,A -85,B 0,C 180,E1 -25532.205,E2 -25532.205} C_VEL
LIN {X 0,Y 145.614,Z 294.295,A -85,B 0,C 180,E1 -25535.211,E2 -25535.211} C_VEL
LIN {X 0,Y 142.98,Z 290.83,A -85,B 0,C 180,E1 -25538.085,E2 -25538.085} C_VEL
LIN {X 0,Y 142.227,Z 289.749,A -85,B 0,C 180,E1 -25539.009,E2 -25539.009} C_VEL
LIN {X 0,Y 139.8,Z 287.032,A -85,B 0,C 180,E1 -25542.257,E2 -25542.257} C_VEL
LIN {X 0,Y 138.686,Z 284.776,A -85,B 0,C 180,E1 -25544.196,E2 -25544.196} C_VEL
LIN {X 0,Y 135.906,Z 282.422,A -85,B 0,C 180,E1 -25549.848,E2 -25549.848} C_VEL
LIN {X 0,Y 134.588,Z 279.56,A -85,B 0,C 180,E1 -25555.509,E2 -25555.509} C_VEL
LIN {X 0,Y 134.296,Z 278.853,A -85,B 0,C 180,E1 -25560.002,E2 -25560.002} C_VEL
LIN {X 0,Y 134.703,Z 279.801,A -85,B 0,C 180,E1 -25564.865,E2 -25564.865} C_VEL
LIN {X 0,Y 137.639,Z 284.222,A -85,B 0,C 180,E1 -25573.661,E2 -25573.661} C_VEL
LIN {X 0,Y 138.801,Z 285.105,A -85,B 0,C 180,E1 -25575.653,E2 -25575.653} C_VEL
LIN {X 0,Y 140.878,Z 288.501,A -85,B 0,C 180,E1 -25578.923,E2 -25578.923} C_VEL
LIN {X 0,Y 142.724,Z 290.386,A -85,B 0,C 180,E1 -25581.214,E2 -25581.214} C_VEL
LIN {X 0,Y 145.29,Z 293.981,A -85,B 0,C 180,E1 -25584.09,E2 -25584.09} C_VEL
LIN {X 0,Y 146.503,Z 295.539,A -85,B 0,C 180,E1 -25585.295,E2 -25585.295} C_VEL
LIN {X 0,Y 149.596,Z 299.953,A -85,B 0,C 180,E1 -25588.118,E2 -25588.118} C_VEL
LIN {X 0,Y 152.576,Z 304.475,A -85,B 0,C 180,E1 -25590.541,E2 -25590.541} C_VEL
LIN {X 0,Y 156.073,Z 311.188,A -85,B 0,C 180,E1 -25593.19,E2 -25593.19} C_VEL
LIN {X 0,Y 159.873,Z 319.682,A -85,B 0,C 180,E1 -25595.844,E2 -25595.844} C_VEL
LIN {X 0,Y 163.359,Z 328.448,A -85,B 0,C 180,E1 -25598.106,E2 -25598.106} C_VEL
LIN {X 0,Y 165.629,Z 335.069,A -85,B 0,C 180,E1 -25599.532,E2 -25599.532} C_VEL
LIN {X 0,Y 163.089,Z 367.411,A -85,B 0,C 180,E1 -25600.752,E2 -25600.752} C_VEL
LIN {X 0,Y 161.172,Z 380.232,A -85,B 0,C 180,E1 -25601.538,E2 -25601.538} C_VEL
LIN {X 0,Y 157.995,Z 393.569,A -85,B 0,C 180,E1 -25602.781,E2 -25602.781} C_VEL
LIN {X 0,Y 155.073,Z 403.079,A -85,B 0,C 180,E1 -25603.99,E2 -25603.99} C_VEL
LIN {X 0,Y 151.685,Z 412.349,A -85,B 0,C 180,E1 -25605.51,E2 -25605.51} C_VEL
LIN {X 0,Y 147.914,Z 421.289,A -85,B 0,C 180,E1 -25607.385,E2 -25607.385} C_VEL
LIN {X 0,Y 143.834,Z 429.813,A -85,B 0,C 180,E1 -25609.653,E2 -25609.653} C_VEL
LIN {X 0,Y 139.984,Z 437.027,A -85,B 0,C 180,E1 -25612.047,E2 -25612.047} C_VEL
LIN {X 0,Y 136.434,Z 443.225,A -85,B 0,C 180,E1 -25614.584,E2 -25614.584} C_VEL
LIN {X 0,Y 132.274,Z 450.178,A -85,B 0,C 180,E1 -25618.227,E2 -25618.227} C_VEL
LIN {X 0,Y 128.377,Z 456.181,A -85,B 0,C 180,E1 -25622.268,E2 -25622.268} C_VEL
LIN {X 0,Y 124.909,Z 461.311,A -85,B 0,C 180,E1 -25626.806,E2 -25626.806} C_VEL
LIN {X 0,Y 122.243,Z 465.302,A -85,B 0,C 180,E1 -25631.566,E2 -25631.566} C_VEL
LIN {X 0,Y 120.523,Z 468.261,A -85,B 0,C 180,E1 -25636.512,E2 -25636.512} C_VEL
LIN {X 0,Y 119.392,Z 470.722,A -85,B 0,C 180,E1 -25643.239,E2 -25643.239} C_VEL
LIN {X 0,Y 119.231,Z 471.318,A -85,B 0,C 180,E1 -25646.621,E2 -25646.621} C_VEL
LIN {X 0,Y 119.337,Z 471.479,A -85,B 0,C 180,E1 -25650,E2 -25650} C_VEL
LIN {X 0,Y 119.221,Z 471.318,A -85,B 0,C 180,E1 -25653.379,E2 -25653.379} C_VEL
LIN {X 0,Y 119.326,Z 470.721,A -85,B 0,C 180,E1 -25656.765,E2 -25656.765} C_VEL
LIN {X 0,Y 120.489,Z 468.26,A -85,B 0,C 180,E1 -25663.492,E2 -25663.492} C_VEL
LIN {X 0,Y 122.243,Z 465.302,A -85,B 0,C 180,E1 -25668.434,E2 -25668.434} C_VEL
LIN {X 0,Y 124.908,Z 461.311,A -85,B 0,C 180,E1 -25673.195,E2 -25673.195} C_VEL
LIN {X 0,Y 128.37,Z 456.181,A -85,B 0,C 180,E1 -25677.733,E2 -25677.733} C_VEL
LIN {X 0,Y 132.215,Z 450.252,A -85,B 0,C 180,E1 -25681.732,E2 -25681.732} C_VEL
LIN {X 0,Y 136.434,Z 443.225,A -85,B 0,C 180,E1 -25685.416,E2 -25685.416} C_VEL
LIN {X 0,Y 141.864,Z 433.648,A -85,B 0,C 180,E1 -25689.171,E2 -25689.171} C_VEL
LIN {X 0,Y 146.361,Z 424.691,A -85,B 0,C 180,E1 -25691.778,E2 -25691.778} C_VEL
LIN {X 0,Y 150.021,Z 416.4,A -85,B 0,C 180,E1 -25693.708,E2 -25693.708} C_VEL
LIN {X 0,Y 153.903,Z 406.34,A -85,B 0,C 180,E1 -25695.522,E2 -25695.522} C_VEL
LIN {X 0,Y 157.091,Z 396.588,A -85,B 0,C 180,E1 -25696.869,E2 -25696.869} C_VEL
LIN {X 0,Y 159.76,Z 386.511,A -85,B 0,C 180,E1 -25697.932,E2 -25697.932} C_VEL
LIN {X 0,Y 161.781,Z 376.53,A -85,B 0,C 180,E1 -25698.716,E2 -25698.716} C_VEL
LIN {X 0,Y 163.247,Z 366.221,A -85,B 0,C 180,E1 -25699.28,E2 -25699.28} C_VEL
LIN {X 0,Y 165.622,Z 335.144,A -85,B 0,C 180,E1 -25700.466,E2 -25700.466} C_VEL
LIN {X 0,Y 163.866,Z 329.997,A -85,B 0,C 180,E1 -25701.564,E2 -25701.564} C_VEL
LIN {X 0,Y 162.369,Z 327.29,A -85,B 0,C 180,E1 -25702.421,E2 -25702.421} C_VEL
LIN {X 0,Y 159.071,Z 324.321,A -85,B 0,C 180,E1 -25704.204,E2 -25704.204} C_VEL
LIN {X 0,Y 155.762,Z 321.589,A -85,B 0,C 180,E1 -25706.135,E2 -25706.135} C_VEL
LIN {X 0,Y 154.212,Z 319.206,A -85,B 0,C 180,E1 -25707.196,E2 -25707.196} C_VEL
LIN {X 0,Y 150.39,Z 310.97,A -85,B 0,C 180,E1 -25710.275,E2 -25710.275} C_VEL
LIN {X 0,Y 146.36,Z 304.645,A -85,B 0,C 180,E1 -25713.82,E2 -25713.82} C_VEL
LIN {X 0,Y 143.487,Z 300.535,A -85,B 0,C 180,E1 -25716.738,E2 -25716.738} C_VEL
LIN {X 0,Y 140.556,Z 296.344,A -85,B 0,C 180,E1 -25720.273,E2 -25720.273} C_VEL
LIN {X 0,Y 137.951,Z 293.063,A -85,B 0,C 180,E1 -25724.106,E2 -25724.106} C_VEL
LIN {X 0,Y 137.198,Z 291.56,A -85,B 0,C 180,E1 -25725.537,E2 -25725.537} C_VEL
LIN {X 0,Y 134.756,Z 289.206,A -85,B 0,C 180,E1 -25730.997,E2 -25730.997} C_VEL
LIN {X 0,Y 133.671,Z 286.536,A -85,B 0,C 180,E1 -25736.23,E2 -25736.23} C_VEL
LIN {X 0,Y 133.432,Z 285.896,A -85,B 0,C 180,E1 -25739.998,E2 -25739.998} C_VEL
LIN {X 0,Y 133.77,Z 286.804,A -85,B 0,C 180,E1 -25744.896,E2 -25744.896} C_VEL
LIN {X 0,Y 136.279,Z 290.972,A -85,B 0,C 180,E1 -25753.151,E2 -25753.151} C_VEL
LIN {X 0,Y 137.387,Z 291.832,A -85,B 0,C 180,E1 -25755.197,E2 -25755.197} C_VEL
LIN {X 0,Y 139.667,Z 295.534,A -85,B 0,C 180,E1 -25758.95,E2 -25758.95} C_VEL
LIN {X 0,Y 141.038,Z 296.997,A -85,B 0,C 180,E1 -25760.735,E2 -25760.735} C_VEL
LIN {X 0,Y 143.643,Z 300.684,A -85,B 0,C 180,E1 -25763.805,E2 -25763.805} C_VEL
LIN {X 0,Y 147.423,Z 306.307,A -85,B 0,C 180,E1 -25767.557,E2 -25767.557} C_VEL
LIN {X 0,Y 151.697,Z 312.977,A -85,B 0,C 180,E1 -25771.135,E2 -25771.135} C_VEL
LIN {X 0,Y 156.497,Z 321.495,A -85,B 0,C 180,E1 -25774.635,E2 -25774.635} C_VEL
LIN {X 0,Y 160.555,Z 329.574,A -85,B 0,C 180,E1 -25777.284,E2 -25777.284} C_VEL
LIN {X 0,Y 164.592,Z 338.804,A -85,B 0,C 180,E1 -25779.728,E2 -25779.728} C_VEL
LIN {X 0,Y 169.134,Z 351.177,A -85,B 0,C 180,E1 -25782.33,E2 -25782.33} C_VEL
LIN {X 0,Y 174.791,Z 365.914,A -85,B 0,C 180,E1 -25785.431,E2 -25785.431} C_VEL
LIN {X 0,Y 179.632,Z 377.412,A -85,B 0,C 180,E1 -25788.309,E2 -25788.309} C_VEL
LIN {X 0,Y 184.833,Z 388.156,A -85,B 0,C 180,E1 -25791.384,E2 -25791.384} C_VEL
LIN {X 0,Y 190.22,Z 397.403,A -85,B 0,C 180,E1 -25794.371,E2 -25794.371} C_VEL
LIN {X 0,Y 196.416,Z 406.306,A -85,B 0,C 180,E1 -25797.54,E2 -25797.54} C_VEL
LIN {X 0,Y 203.405,Z 414.601,A -85,B 0,C 180,E1 -25800.764,E2 -25800.764} C_VEL
LIN {X 0,Y 211.206,Z 422.145,A -85,B 0,C 180,E1 -25803.951,E2 -25803.951} C_VEL
LIN {X 0,Y 220.849,Z 429.501,A -85,B 0,C 180,E1 -25807.344,E2 -25807.344} C_VEL
LIN {X 0,Y 233.823,Z 437.221,A -85,B 0,C 180,E1 -25811.222,E2 -25811.222} C_VEL
LIN {X 0,Y 247.542,Z 443.876,A -85,B 0,C 180,E1 -25814.858,E2 -25814.858} C_VEL
LIN {X 0,Y 258.832,Z 448.924,A -85,B 0,C 180,E1 -25817.818,E2 -25817.818} C_VEL
LIN {X 0,Y 267.149,Z 452.689,A -85,B 0,C 180,E1 -25820.233,E2 -25820.233} C_VEL
LIN {X 0,Y 270.235,Z 454.071,A -85,B 0,C 180,E1 -25821.208,E2 -25821.208} C_VEL
LIN {X 0,Y 274.117,Z 455.916,A -85,B 0,C 180,E1 -25822.635,E2 -25822.635} C_VEL
LIN {X 0,Y 277.378,Z 457.621,A -85,B 0,C 180,E1 -25824.183,E2 -25824.183} C_VEL
LIN {X 0,Y 281.62,Z 459.539,A -85,B 0,C 180,E1 -25826.569,E2 -25826.569} C_VEL
LIN {X 0,Y 282.43,Z 459.854,A -85,B 0,C 180,E1 -25827.147,E2 -25827.147} C_VEL
LIN {X 0,Y 283.873,Z 460.412,A -85,B 0,C 180,E1 -25828.581,E2 -25828.581} C_VEL
LIN {X 0,Y 284.644,Z 460.595,A -85,B 0,C 180,E1 -25830,E2 -25830} C_VEL
LIN {X 0,Y 283.886,Z 460.411,A -85,B 0,C 180,E1 -25831.419,E2 -25831.419} C_VEL
LIN {X 0,Y 282.435,Z 459.855,A -85,B 0,C 180,E1 -25832.853,E2 -25832.853} C_VEL
LIN {X 0,Y 280.089,Z 458.927,A -85,B 0,C 180,E1 -25834.317,E2 -25834.317} C_VEL
LIN {X 0,Y 275.896,Z 456.837,A -85,B 0,C 180,E1 -25836.564,E2 -25836.564} C_VEL
LIN {X 0,Y 274.14,Z 455.915,A -85,B 0,C 180,E1 -25837.365,E2 -25837.365} C_VEL
LIN {X 0,Y 269.602,Z 453.791,A -85,B 0,C 180,E1 -25838.998,E2 -25838.998} C_VEL
LIN {X 0,Y 261.339,Z 450.072,A -85,B 0,C 180,E1 -25841.479,E2 -25841.479} C_VEL
LIN {X 0,Y 253.138,Z 446.443,A -85,B 0,C 180,E1 -25843.662,E2 -25843.662} C_VEL
LIN {X 0,Y 241.978,Z 441.29,A -85,B 0,C 180,E1 -25846.578,E2 -25846.578} C_VEL
LIN {X 0,Y 228.686,Z 434.427,A -85,B 0,C 180,E1 -25850.226,E2 -25850.226} C_VEL
LIN {X 0,Y 215.948,Z 426.015,A -85,B 0,C 180,E1 -25854.323,E2 -25854.323} C_VEL
LIN {X 0,Y 206.666,Z 418.011,A -85,B 0,C 180,E1 -25857.853,E2 -25857.853} C_VEL
LIN {X 0,Y 198.123,Z 408.498,A -85,B 0,C 180,E1 -25861.644,E2 -25861.644} C_VEL
LIN {X 0,Y 191.357,Z 399.19,A -85,B 0,C 180,E1 -25865.022,E2 -25865.022} C_VEL
LIN {X 0,Y 186.473,Z 391.222,A -85,B 0,C 180,E1 -25867.679,E2 -25867.679} C_VEL
LIN {X 0,Y 182.008,Z 382.379,A -85,B 0,C 180,E1 -25870.307,E2 -25870.307} C_VEL
LIN {X 0,Y 177.456,Z 372.337,A -85,B 0,C 180,E1 -25872.995,E2 -25872.995} C_VEL
LIN {X 0,Y 173.074,Z 361.574,A -85,B 0,C 180,E1 -25875.537,E2 -25875.537} C_VEL
LIN {X 0,Y 166.641,Z 344.115,A -85,B 0,C 180,E1 -25879.081,E2 -25879.081} C_VEL
LIN {X 0,Y 161.708,Z 331.925,A -85,B 0,C 180,E1 -25882.012,E2 -25882.012} C_VEL
LIN {X 0,Y 156.601,Z 321.689,A -85,B 0,C 180,E1 -25885.294,E2 -25885.294} C_VEL
LIN {X 0,Y 151.696,Z 312.987,A -85,B 0,C 180,E1 -25888.865,E2 -25888.865} C_VEL
LIN {X 0,Y 148.336,Z 307.743,A -85,B 0,C 180,E1 -25891.625,E2 -25891.625} C_VEL
LIN {X 0,Y 145.903,Z 304.092,A -85,B 0,C 180,E1 -25893.863,E2 -25893.863} C_VEL
LIN {X 0,Y 143.486,Z 300.517,A -85,B 0,C 180,E1 -25896.359,E2 -25896.359} C_VEL
LIN {X 0,Y 140.999,Z 296.927,A -85,B 0,C 180,E1 -25899.317,E2 -25899.317} C_VEL
LIN {X 0,Y 137.95,Z 293.047,A -85,B 0,C 180,E1 -25903.729,E2 -25903.729} C_VEL
LIN {X 0,Y 137.2,Z 291.514,A -85,B 0,C 180,E1 -25905.162,E2 -25905.162} C_VEL
LIN {X 0,Y 134.731,Z 289.178,A -85,B 0,C 180,E1 -25910.689,E2 -25910.689} C_VEL
LIN {X 0,Y 133.719,Z 286.654,A -85,B 0,C 180,E1 -25915.48,E2 -25915.48} C_VEL
LIN {X 0,Y 133.432,Z 285.896,A -85,B 0,C 180,E1 -25920.002,E2 -25920.002} C_VEL
LIN {X 0,Y 133.795,Z 286.913,A -85,B 0,C 180,E1 -25924.71,E2 -25924.71} C_VEL
LIN {X 0,Y 136.412,Z 291.057,A -85,B 0,C 180,E1 -25933.028,E2 -25933.028} C_VEL
LIN {X 0,Y 137.433,Z 291.958,A -85,B 0,C 180,E1 -25934.911,E2 -25934.911} C_VEL
LIN {X 0,Y 139.765,Z 295.613,A -85,B 0,C 180,E1 -25938.699,E2 -25938.699} C_VEL
LIN {X 0,Y 141.015,Z 296.966,A -85,B 0,C 180,E1 -25940.325,E2 -25940.325} C_VEL
LIN {X 0,Y 143.804,Z 300.845,A -85,B 0,C 180,E1 -25943.589,E2 -25943.589} C_VEL
LIN {X 0,Y 147.462,Z 306.371,A -85,B 0,C 180,E1 -25947.211,E2 -25947.211} C_VEL
LIN {X 0,Y 150.489,Z 311.201,A -85,B 0,C 180,E1 -25949.812,E2 -25949.812} C_VEL
LIN {X 0,Y 154.173,Z 319.131,A -85,B 0,C 180,E1 -25952.775,E2 -25952.775} C_VEL
LIN {X 0,Y 158.712,Z 330.386,A -85,B 0,C 180,E1 -25956.074,E2 -25956.074} C_VEL
LIN {X 0,Y 161.008,Z 337.331,A -85,B 0,C 180,E1 -25957.671,E2 -25957.671} C_VEL
LIN {X 0,Y 158.552,Z 367.225,A -85,B 0,C 180,E1 -25958.81,E2 -25958.81} C_VEL
LIN {X 0,Y 156.47,Z 380.56,A -85,B 0,C 180,E1 -25959.633,E2 -25959.633} C_VEL
LIN {X 0,Y 153.27,Z 393.377,A -85,B 0,C 180,E1 -25960.836,E2 -25960.836} C_VEL
LIN {X 0,Y 150.221,Z 402.886,A -85,B 0,C 180,E1 -25962.038,E2 -25962.038} C_VEL
LIN {X 0,Y 146.7,Z 412.157,A -85,B 0,C 180,E1 -25963.565,E2 -25963.565} C_VEL
LIN {X 0,Y 142.765,Z 421.096,A -85,B 0,C 180,E1 -25965.453,E2 -25965.453} C_VEL
LIN {X 0,Y 138.481,Z 429.619,A -85,B 0,C 180,E1 -25967.744,E2 -25967.744} C_VEL
LIN {X 0,Y 134.452,Z 436.834,A -85,B 0,C 180,E1 -25970.184,E2 -25970.184} C_VEL
LIN {X 0,Y 130.692,Z 443.032,A -85,B 0,C 180,E1 -25972.773,E2 -25972.773} C_VEL
LIN {X 0,Y 126.534,Z 449.57,A -85,B 0,C 180,E1 -25976.26,E2 -25976.26} C_VEL
LIN {X 0,Y 123.563,Z 454.074,A -85,B 0,C 180,E1 -25979.21,E2 -25979.21} C_VEL
LIN {X 0,Y 119.542,Z 459.564,A -85,B 0,C 180,E1 -25983.837,E2 -25983.837} C_VEL
LIN {X 0,Y 116.338,Z 463.89,A -85,B 0,C 180,E1 -25988.749,E2 -25988.749} C_VEL
LIN {X 0,Y 114.771,Z 466.262,A -85,B 0,C 180,E1 -25992.171,E2 -25992.171} C_VEL
LIN {X 0,Y 113.614,Z 468.068,A -85,B 0,C 180,E1 -25995.674,E2 -25995.674} C_VEL
LIN {X 0,Y 112.314,Z 470.529,A -85,B 0,C 180,E1 -26002.811,E2 -26002.811} C_VEL
LIN {X 0,Y 112.139,Z 471.125,A -85,B 0,C 180,E1 -26006.407,E2 -26006.407} C_VEL
LIN {X 0,Y 112.253,Z 471.286,A -85,B 0,C 180,E1 -26010,E2 -26010} C_VEL
LIN {X 0,Y 112.129,Z 471.125,A -85,B 0,C 180,E1 -26013.594,E2 -26013.594} C_VEL
LIN {X 0,Y 112.262,Z 470.527,A -85,B 0,C 180,E1 -26017.193,E2 -26017.193} C_VEL
LIN {X 0,Y 113.571,Z 468.067,A -85,B 0,C 180,E1 -26024.331,E2 -26024.331} C_VEL
LIN {X 0,Y 115.494,Z 465.108,A -85,B 0,C 180,E1 -26029.553,E2 -26029.553} C_VEL
LIN {X 0,Y 118.398,Z 461.118,A -85,B 0,C 180,E1 -26034.552,E2 -26034.552} C_VEL
LIN {X 0,Y 122.118,Z 455.988,A -85,B 0,C 180,E1 -26039.287,E2 -26039.287} C_VEL
LIN {X 0,Y 125.805,Z 450.642,A -85,B 0,C 180,E1 -26043.071,E2 -26043.071} C_VEL
LIN {X 0,Y 129.805,Z 444.407,A -85,B 0,C 180,E1 -26046.553,E2 -26046.553} C_VEL
LIN {X 0,Y 133.477,Z 438.459,A -85,B 0,C 180,E1 -26049.186,E2 -26049.186} C_VEL
LIN {X 0,Y 137.434,Z 431.537,A -85,B 0,C 180,E1 -26051.666,E2 -26051.666} C_VEL
LIN {X 0,Y 141.669,Z 423.364,A -85,B 0,C 180,E1 -26053.989,E2 -26053.989} C_VEL
LIN {X 0,Y 145.53,Z 414.857,A -85,B 0,C 180,E1 -26055.918,E2 -26055.918} C_VEL
LIN {X 0,Y 149.022,Z 406.147,A -85,B 0,C 180,E1 -26057.467,E2 -26057.467} C_VEL
LIN {X 0,Y 152.326,Z 396.395,A -85,B 0,C 180,E1 -26058.818,E2 -26058.818} C_VEL
LIN {X 0,Y 155.099,Z 386.318,A -85,B 0,C 180,E1 -26059.876,E2 -26059.876} C_VEL
LIN {X 0,Y 157.15,Z 376.575,A -85,B 0,C 180,E1 -26060.643,E2 -26060.643} C_VEL
LIN {X 0,Y 158.646,Z 366.516,A -85,B 0,C 180,E1 -26061.203,E2 -26061.203} C_VEL
LIN {X 0,Y 161.004,Z 337.376,A -85,B 0,C 180,E1 -26062.328,E2 -26062.328} C_VEL
LIN {X 0,Y 157.438,Z 327.02,A -85,B 0,C 180,E1 -26064.822,E2 -26064.822} C_VEL
LIN {X 0,Y 154.212,Z 319.206,A -85,B 0,C 180,E1 -26067.196,E2 -26067.196} C_VEL
LIN {X 0,Y 152.084,Z 315.646,A -85,B 0,C 180,E1 -26068.767,E2 -26068.767} C_VEL
LIN {X 0,Y 149.637,Z 313.078,A -85,B 0,C 180,E1 -26070.579,E2 -26070.579} C_VEL
LIN {X 0,Y 141.753,Z 307.117,A -85,B 0,C 180,E1 -26077.547,E2 -26077.547} C_VEL
LIN {X 0,Y 138.848,Z 302.889,A -85,B 0,C 180,E1 -26081.269,E2 -26081.269} C_VEL
LIN {X 0,Y 136.288,Z 299.214,A -85,B 0,C 180,E1 -26085.439,E2 -26085.439} C_VEL
LIN {X 0,Y 135.75,Z 298.303,A -85,B 0,C 180,E1 -26086.526,E2 -26086.526} C_VEL
LIN {X 0,Y 133.361,Z 295.472,A -85,B 0,C 180,E1 -26092.808,E2 -26092.808} C_VEL
LIN {X 0,Y 132.715,Z 293.438,A -85,B 0,C 180,E1 -26096.963,E2 -26096.963} C_VEL
LIN {X 0,Y 132.567,Z 292.935,A -85,B 0,C 180,E1 -26099.998,E2 -26099.998} C_VEL
LIN {X 0,Y 132.842,Z 293.821,A -85,B 0,C 180,E1 -26104.55,E2 -26104.55} C_VEL
LIN {X 0,Y 135.195,Z 297.927,A -85,B 0,C 180,E1 -26112.762,E2 -26112.762} C_VEL
LIN {X 0,Y 136.091,Z 298.764,A -85,B 0,C 180,E1 -26114.532,E2 -26114.532} C_VEL
LIN {X 0,Y 138.271,Z 302.324,A -85,B 0,C 180,E1 -26118.311,E2 -26118.311} C_VEL
LIN {X 0,Y 139.452,Z 303.761,A -85,B 0,C 180,E1 -26119.955,E2 -26119.955} C_VEL
LIN {X 0,Y 142.592,Z 308.467,A -85,B 0,C 180,E1 -26123.798,E2 -26123.798} C_VEL
LIN {X 0,Y 145.477,Z 312.935,A -85,B 0,C 180,E1 -26126.763,E2 -26126.763} C_VEL
LIN {X 0,Y 149.805,Z 320.131,A -85,B 0,C 180,E1 -26130.577,E2 -26130.577} C_VEL
LIN {X 0,Y 154.7,Z 329.465,A -85,B 0,C 180,E1 -26134.304,E2 -26134.304} C_VEL
LIN {X 0,Y 159.389,Z 339.828,A -85,B 0,C 180,E1 -26137.48,E2 -26137.48} C_VEL
LIN {X 0,Y 163.772,Z 351.797,A -85,B 0,C 180,E1 -26140.255,E2 -26140.255} C_VEL
